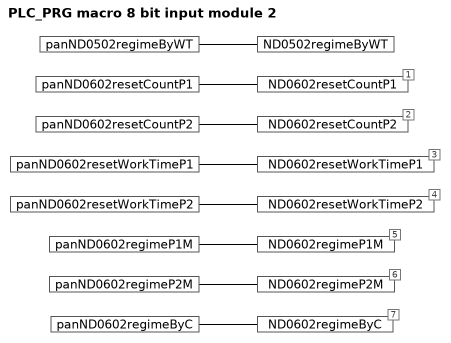
[picture p72: PLC_PRG macro 8 bit input module 2 (CFC)]
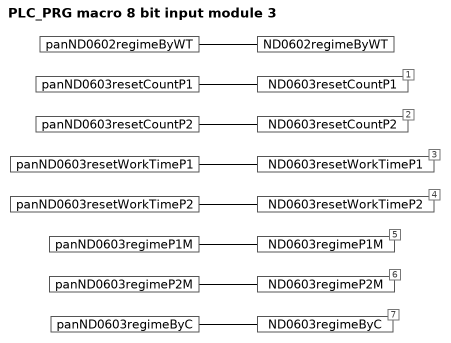
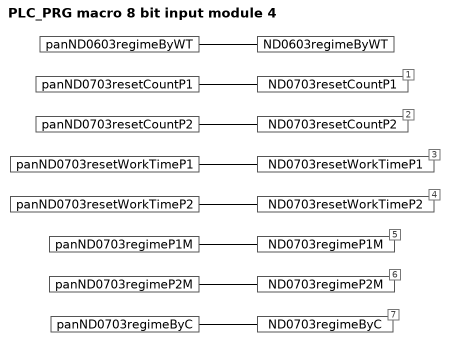
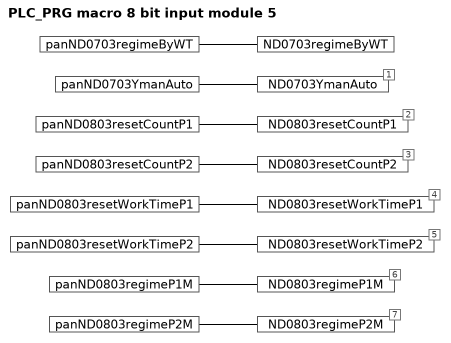
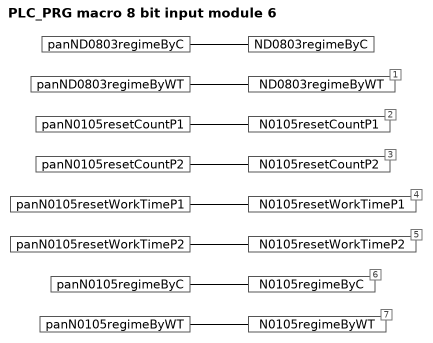
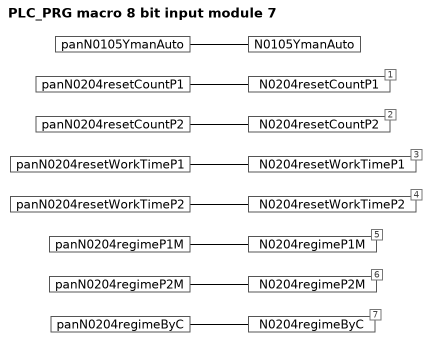
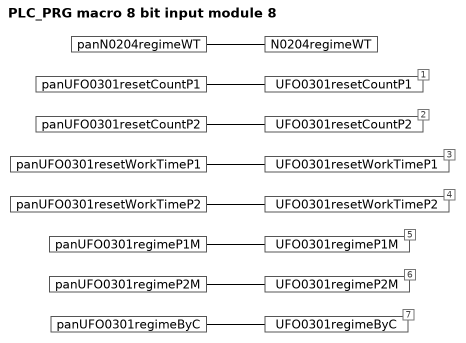
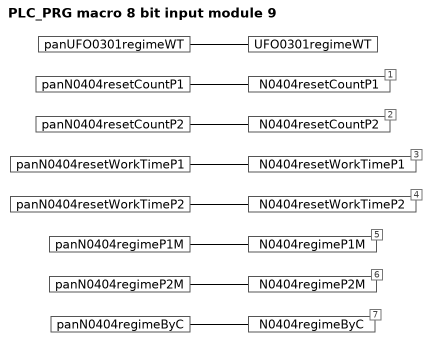
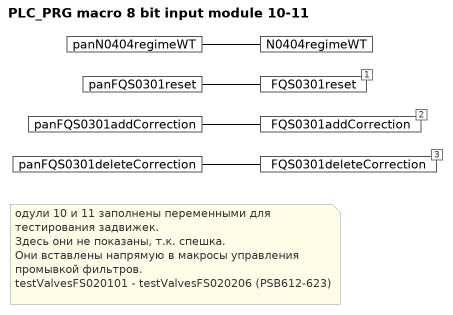
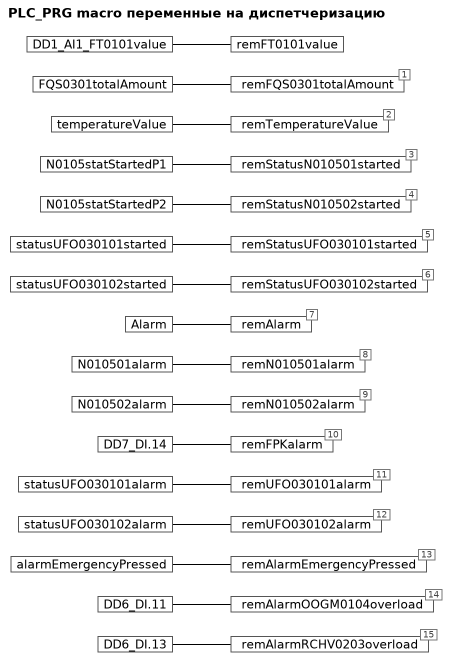
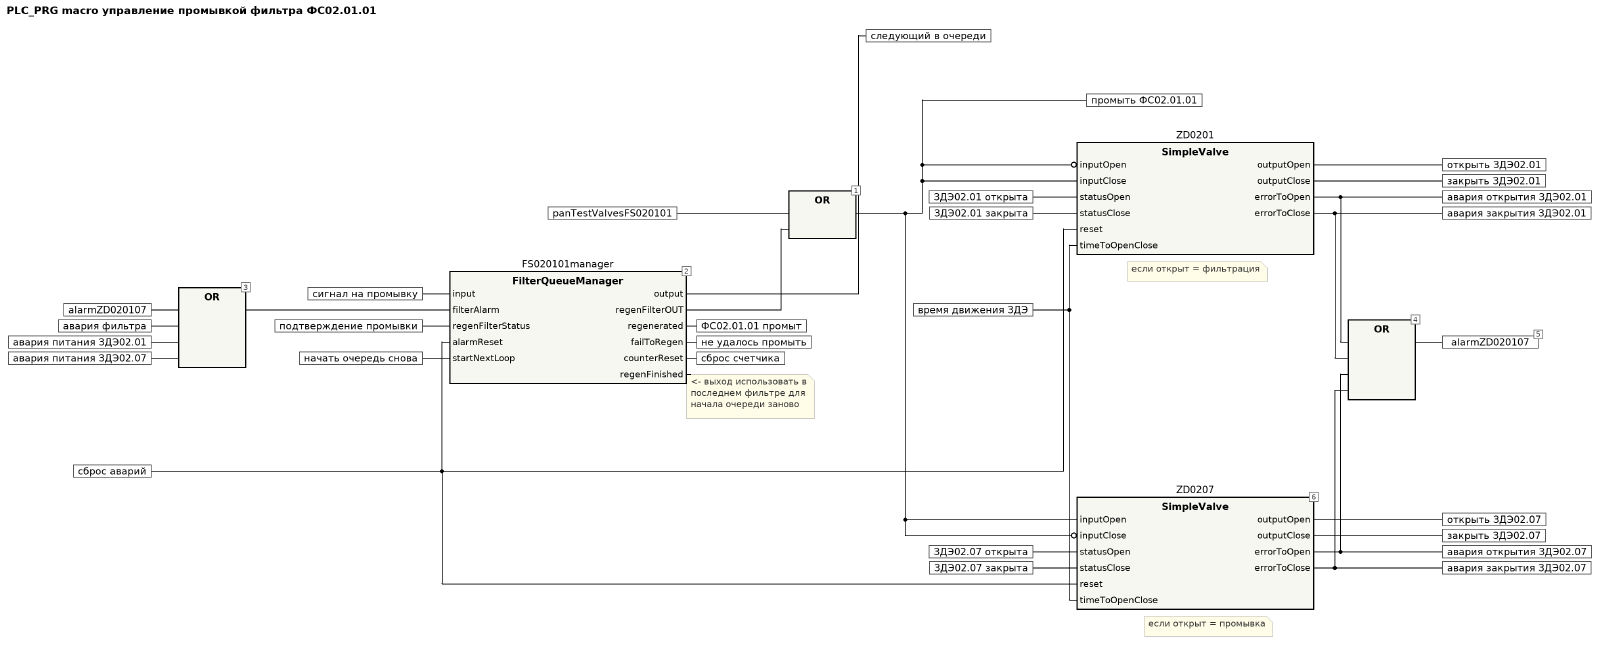
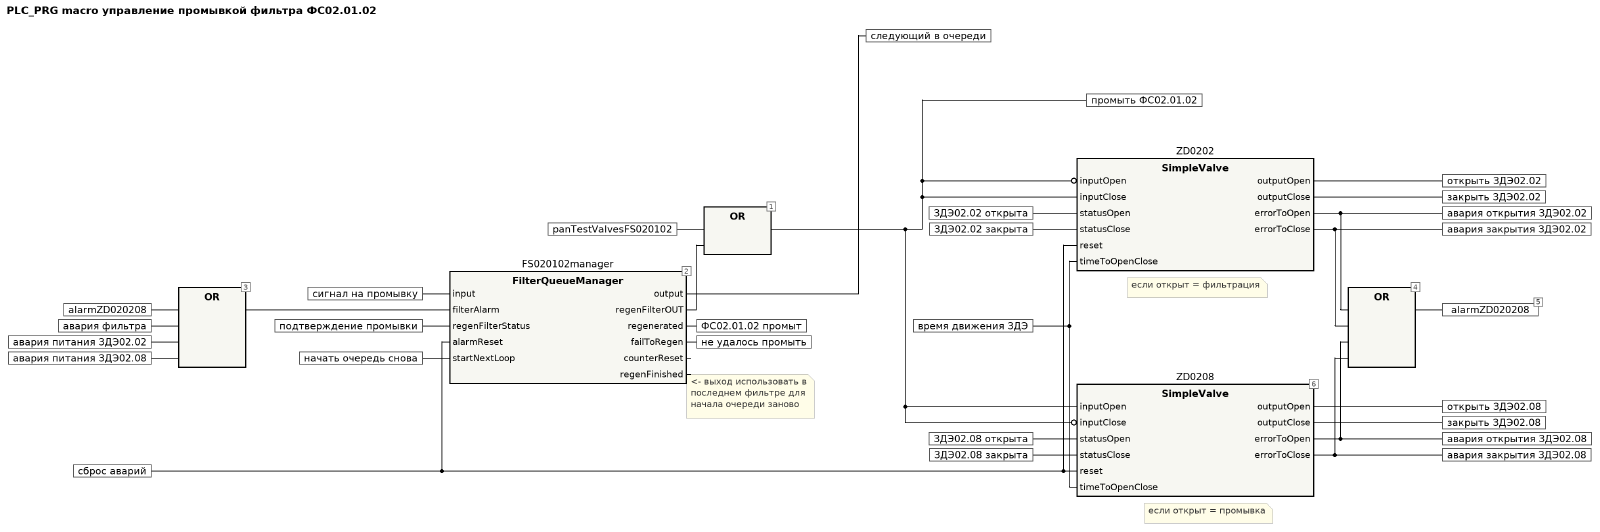
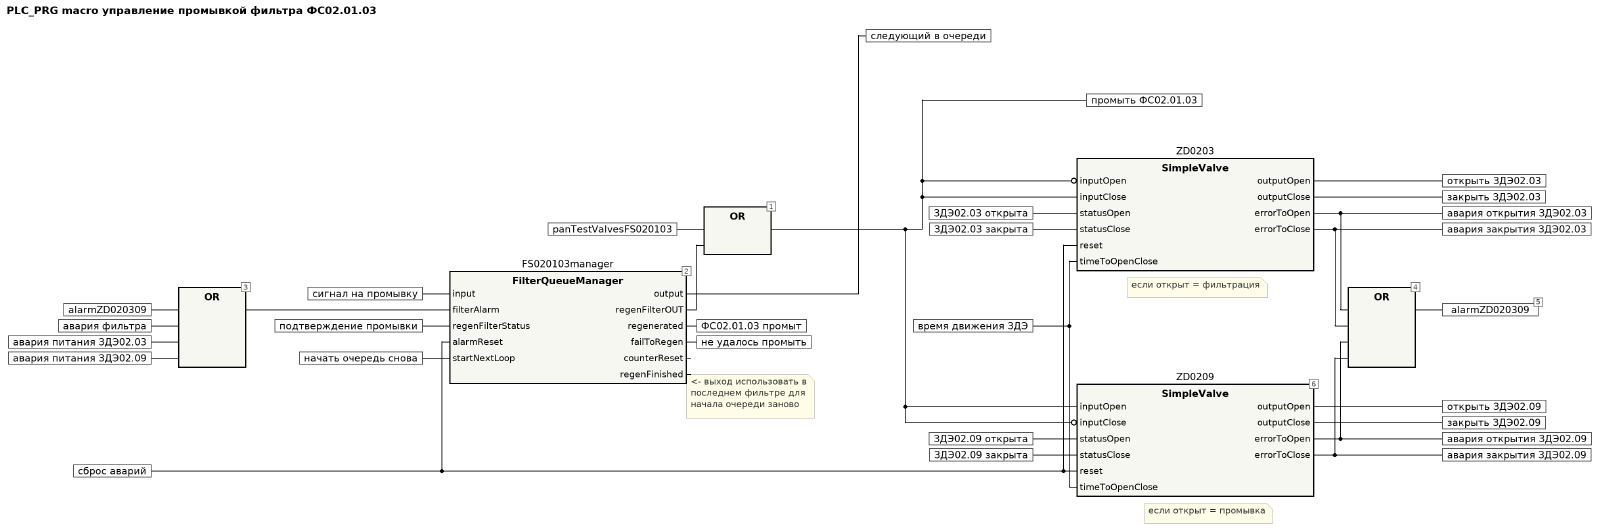
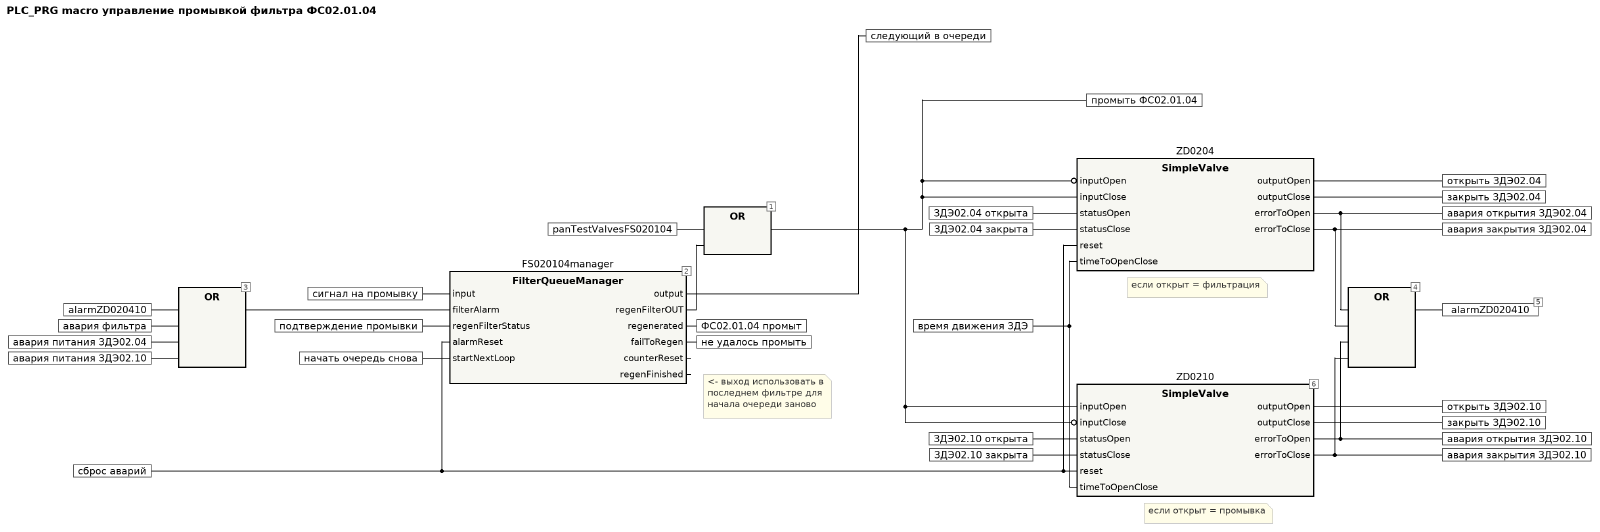
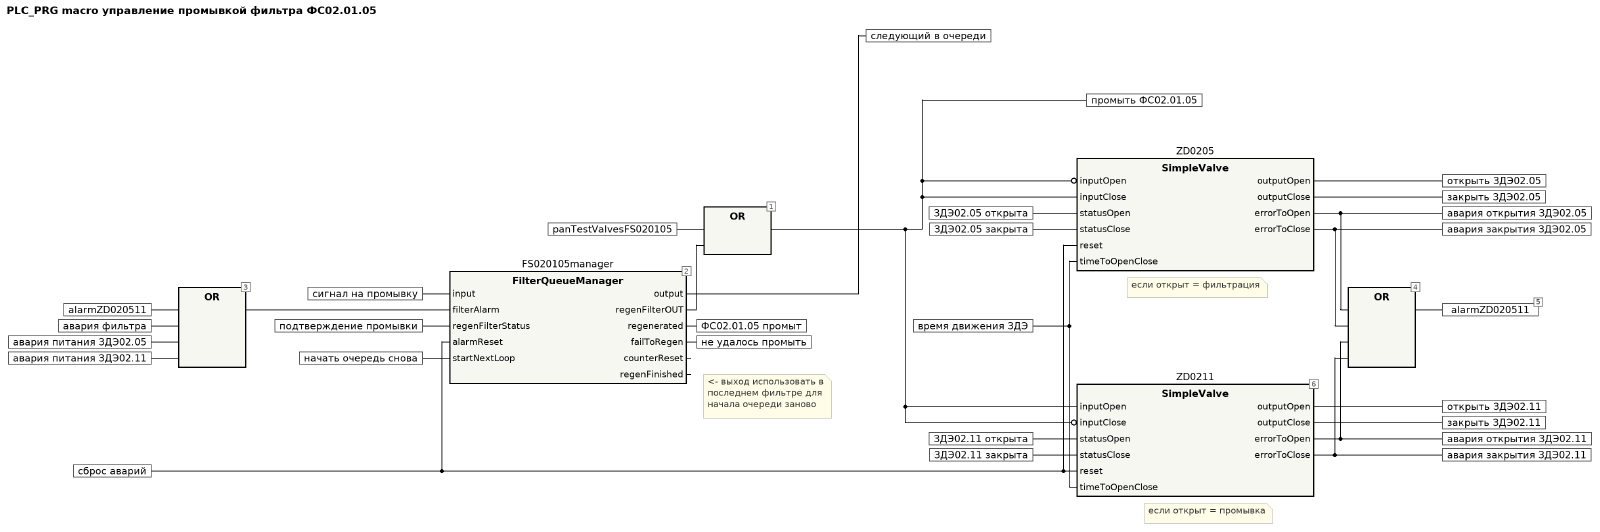
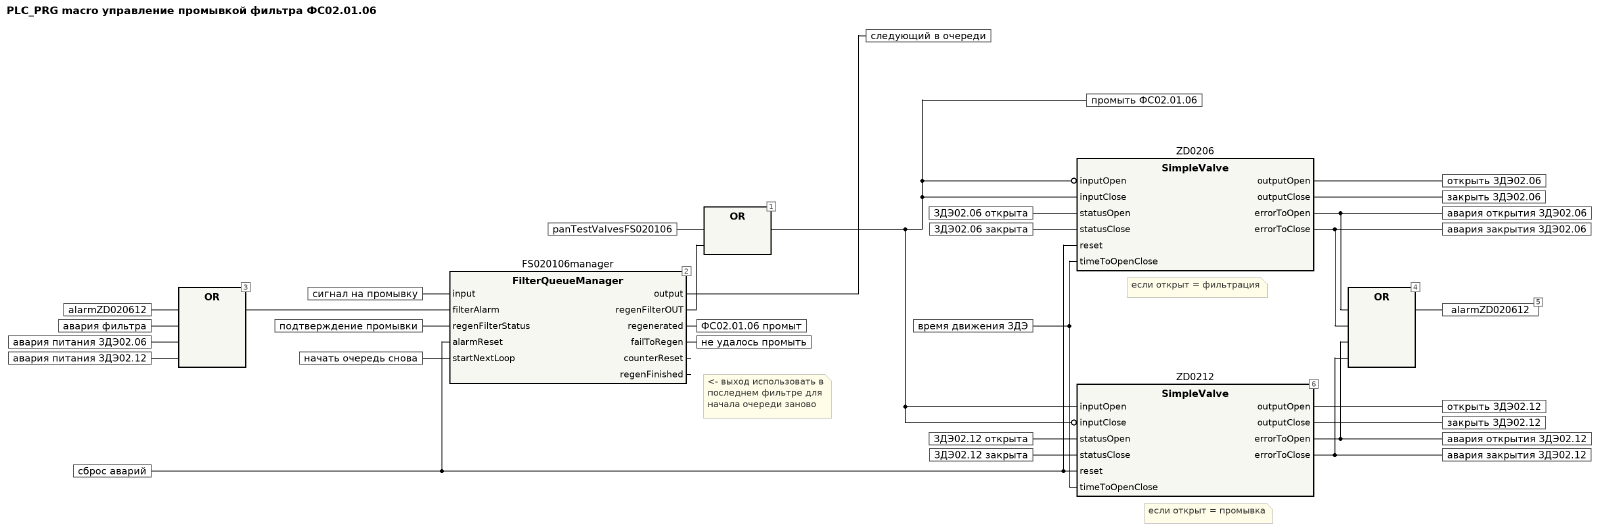
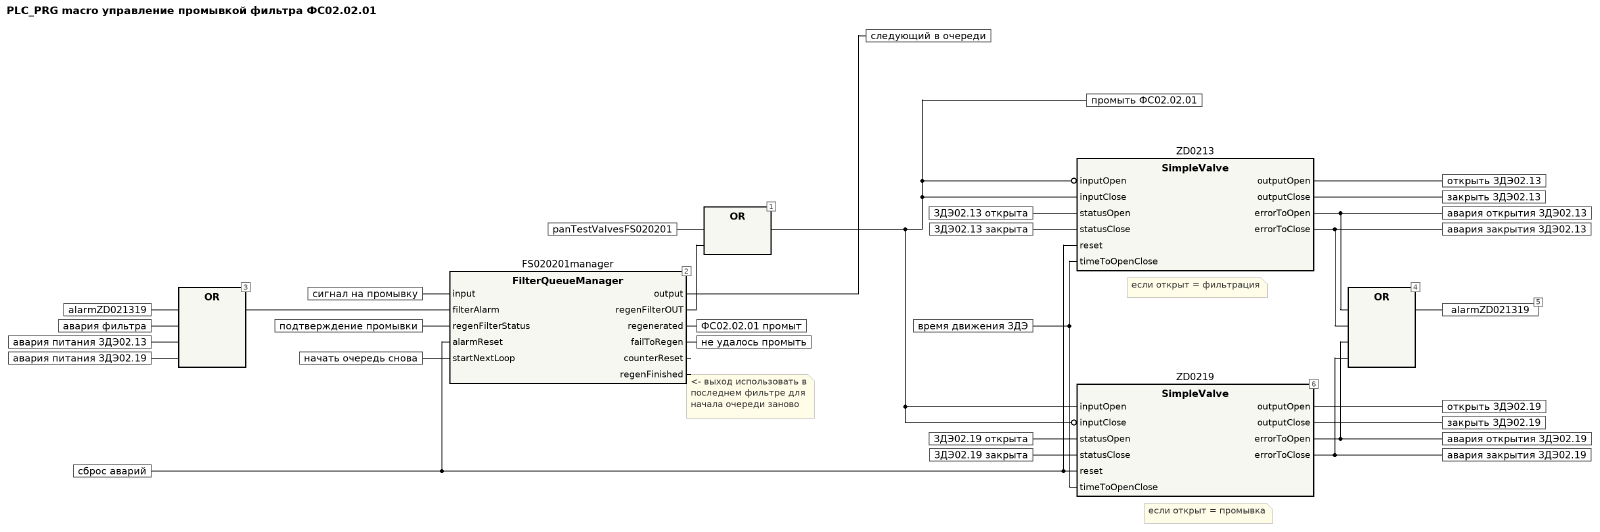
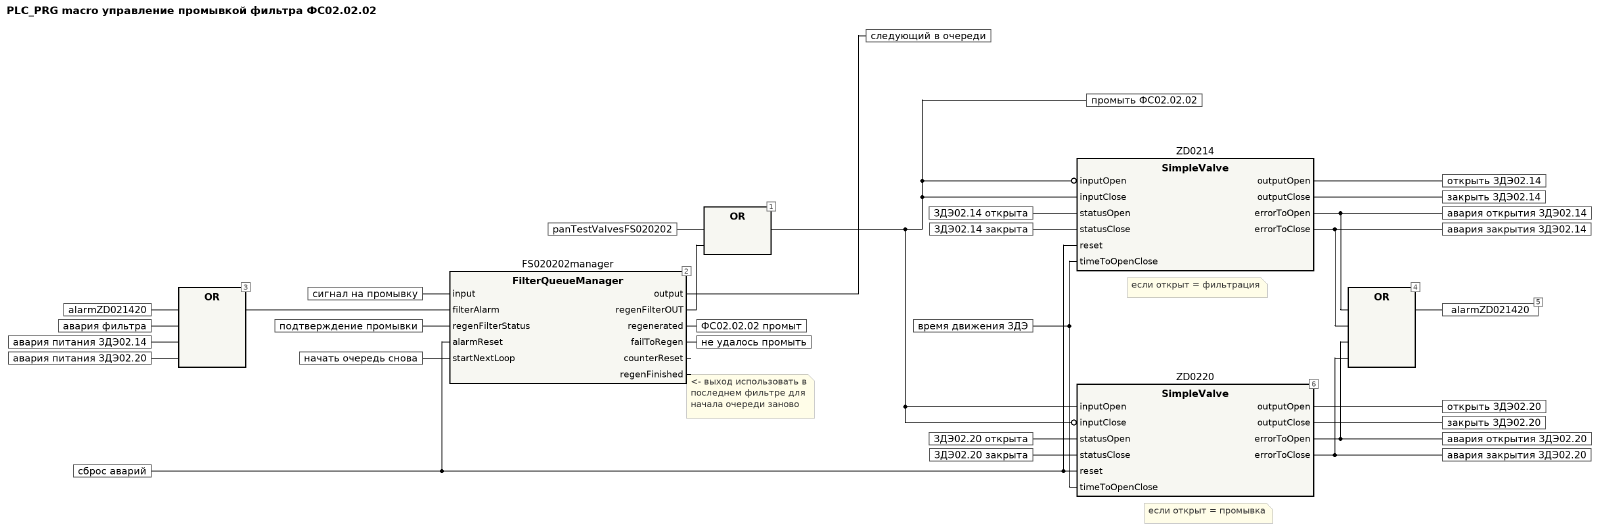
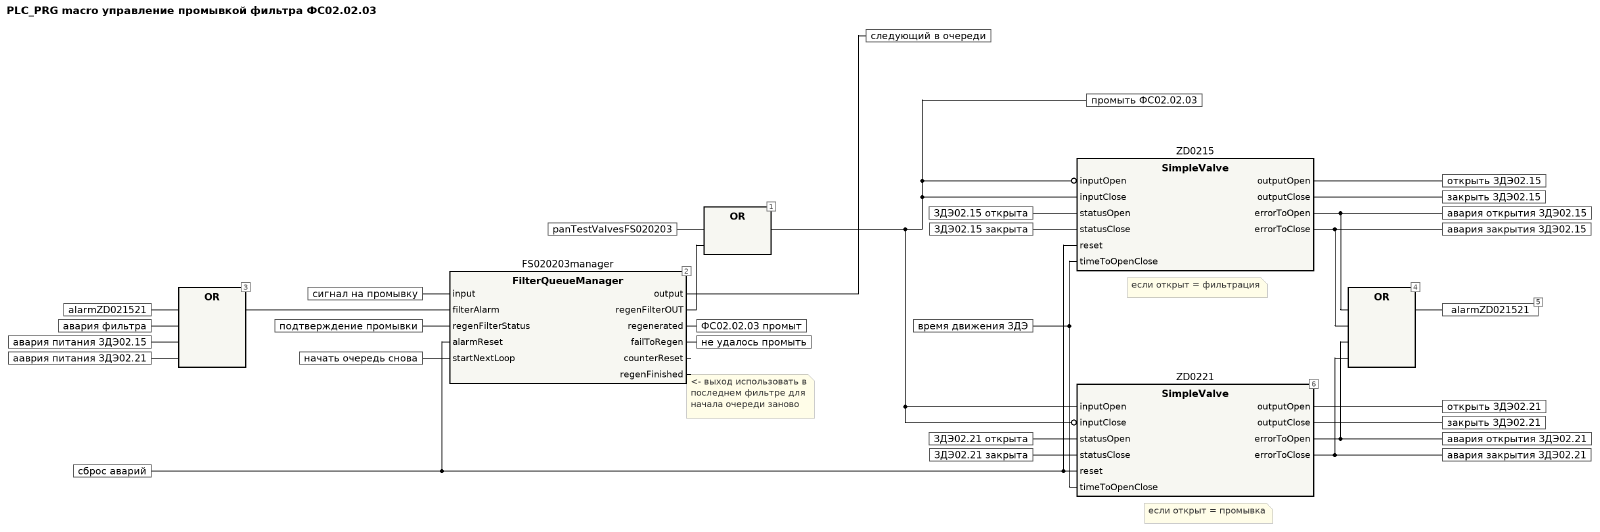
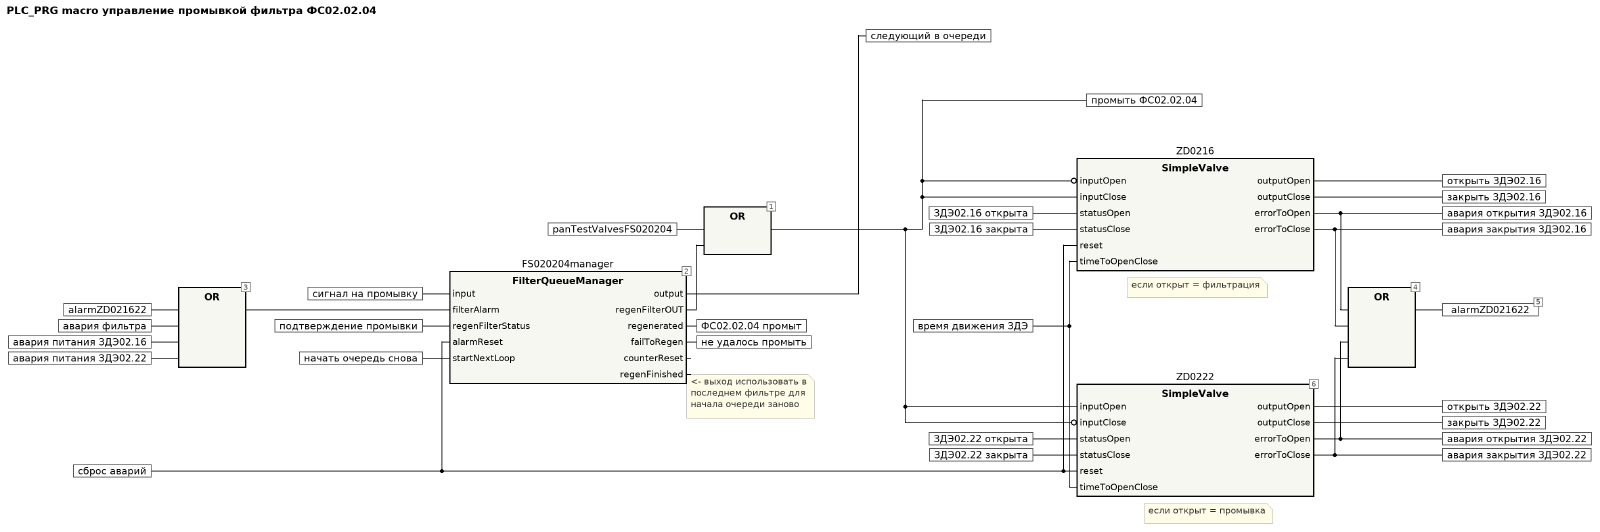
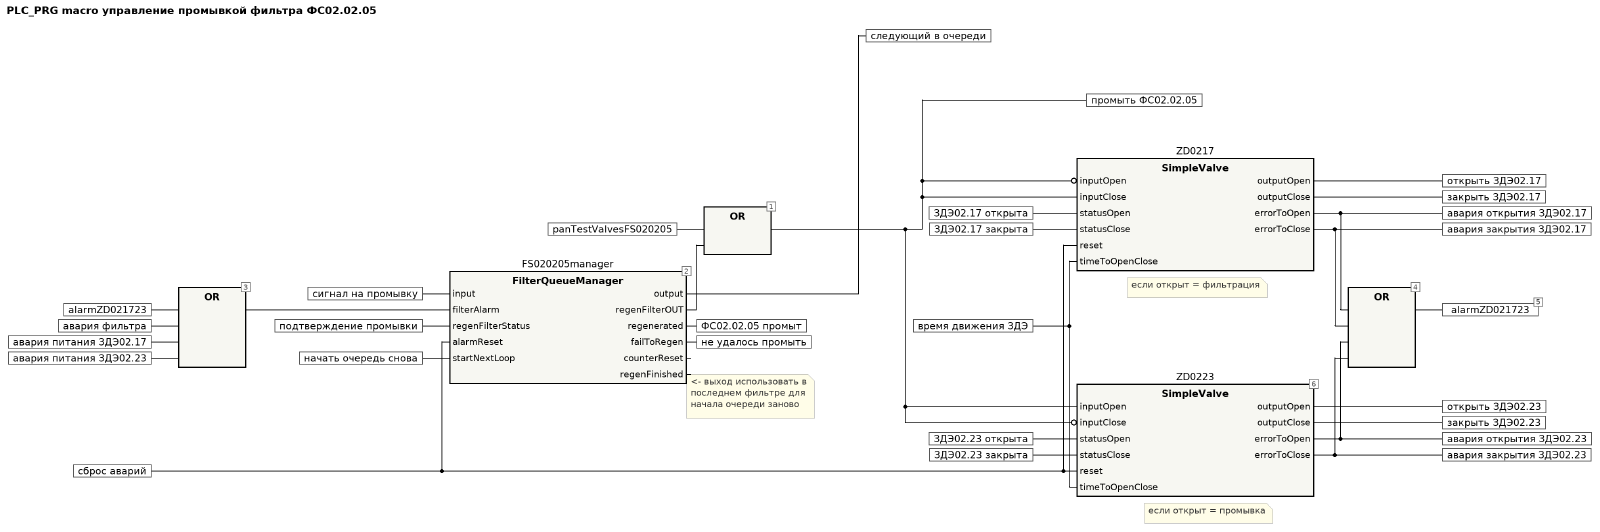
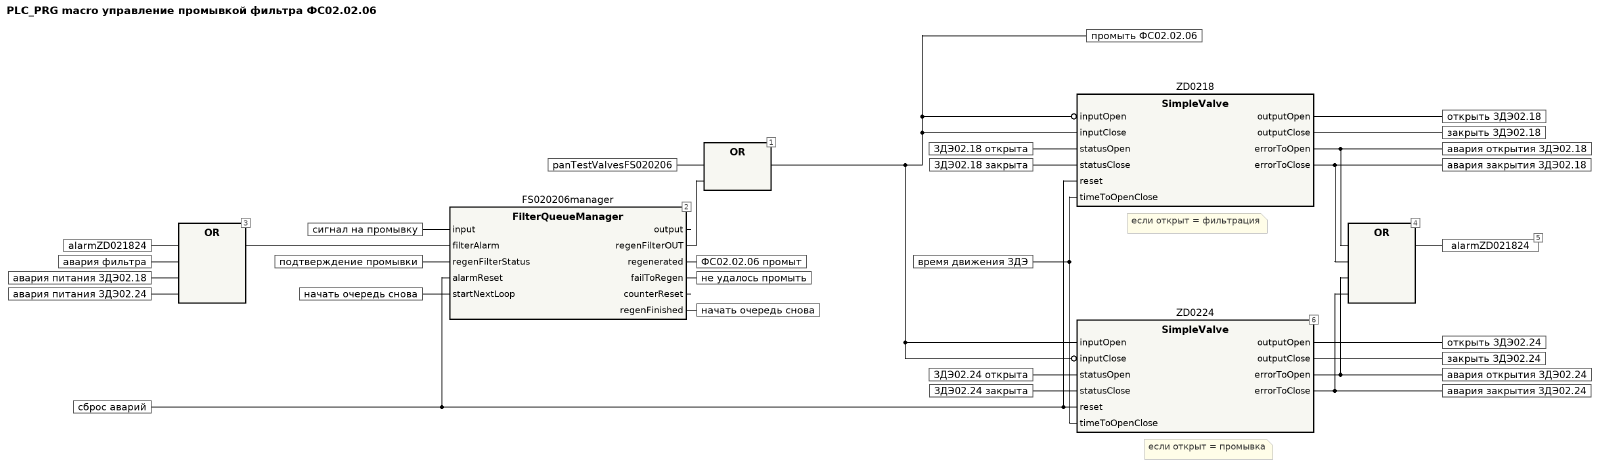
_CFC_ (* Continuous Function Chart, elements in execution order *)
(* в этом макросе лежит управление режимом тестирования задвижек ЗДЭ03 / Тестирование запрещает автоматический запуск УФО от ПЛК *)
(* 1=открыть; 0 = закрыть *)
(* авария питания КШЭ04.01 *)
(* авария НД05.02/02 *)
(* авария НД05.02/01 *)
(* инвертирование сигнала, чтобы все аварии / обозначались как 1 (TRUE) *)
(* авария питания ЗДЭ02.24 *)
(* авария питания ЗДЭ02.23 *)
(* авария питания ЗДЭ02.22 *)
(* авария питания ЗДЭ02.21 *)
(* авария питания ЗДЭ02.20 *)
(* авария питания ЗДЭ02.19 *)
(* авария питания ЗДЭ02.18 *)
(* авария питания ЗДЭ02.17 *)
(* авария питания ЗДЭ02.16 *)
(* авария питания ЗДЭ02.15 *)
(* авария питания ЗДЭ02.14 *)
(* авария питания ЗДЭ02.13 *)
(* авария питания ЗДЭ02.12 *)
(* авария питания ЗДЭ02.11 *)
(* авария питания ЗДЭ02.10 *)
(* авария питания ЗДЭ02.09 *)
(* авария питания ЗДЭ02.08 *)
(* авария питания ЗДЭ02.07 *)
(* авария питания ЗДЭ02.06 *)
(* авария питания ЗДЭ02.05 *)
(* авария питания ЗДЭ02.04 *)
(* авария питания ЗДЭ02.03 *)
(* авария питания ЗДЭ02.02 *)
(* авария питания ЗДЭ02.01 *)
(* очередь передается на 2 ступень *)
(* подсчет общего объема стоков, прошедшего через расходомер FT01.02 *)
(* сброс счетчика стоков до следующей промывки *)
(* авария (при 0) ФС02.02/01 *)
(* авария (при 0) ФС02.02/02 *)
(* авария (при 0) ФС02.02/03 *)
(* авария (при 0) ФС02.02/04 *)
(* авария (при 0) ФС02.02/05 *)
(* авария (при 0) ФС02.02/06 *)
(* авария (при 0) ФС02.01/01 *)
(* авария (при 0) ФС02.01/02 *)
(* авария (при 0) ФС02.01/03 *)
(* авария (при 0) ФС02.01/04 *)
(* авария (при 0) ФС02.01/05 *)
(* авария (при 0) ФС02.01/06 *)
(* 0=авария *)
(* заданный до промывки объем *)
(* текущий объем *)
(* Пуск Н02.04/02 *)
(* Пуск Н02.04/01 *)
(* Стоп Н02.04, / сброс самоподхвата реле, / если активно - пуск невозможен *)
(* Сухой ход Н02.04 (LS02.03) 0=сух.ход *)
(* Клапан КЭМ08.01 открыт. *)
(* Клапан КЭМ07.01 открыт. *)
(* Клапан КЭМ06.01 открыт. *)
(* Клапан КЭМ05.01 открыт. *)
(* промывка ФС02.02/01 *)
(* промывка ФС02.02/02 *)
(* промывка ФС02.02/03 *)
(* промывка ФС02.02/04 *)
(* промывка ФС02.02/05 *)
(* промывка ФС02.02/06 *)
(* Авария Н02.04/02 (0=авария) *)
(* Авария Н02.04/01 (0=авария) *)
(* импульсный расходомер *)
(* авария Н04.04/02, 0=авария *)
(* авария Н04.04/01, 0=авария *)
(* сухой ход Н04.04, 0=защита *)
(* авт.пуск Н04.04 *)
(* пуск Н04.04/01 *)
(* пуск Н04.04/02 *)
(* стоп Н04.04 *)
(* подающий насос ФПК работает *)
(* статус КШЭ04.01 закрыт *)
(* Закрыть КШЭ04.01 *)
(* статус КШЭ04.01 открыт *)
(* Открыть КШЭ04.01 *)
(* авария ФПК *)
(* Авария входа AI6 ПЛК, давл.ФПК *)
(* Давление на входе ФПК / 0...16 бар (мах допуст.10) *)
(* LSА02.01 Перелив РЧВ02.03 *)
(* авария питания ЗДЭ02.25 *)
(* термоконтакт Н01.05/02 *)
(* термоконтакт Н01.05/01 *)
(* Авария ЧРП Н01.05 *)
(* КМ3 питание насоса 2 *)
(* КМ2 питание насоса 1 *)
(* КМ1 питание ЧРП *)
(* Пуск  Н01.05 *)
(* время на создание потока *)
(* Стоп  Н01.05 (сброс самоподхвата реле) *)
(* SA1 Ручной выбор Н01.05/02 = главный *)
(* SA1 Ручной выбор Н01.05/01 = главный *)
(* LS01.04 - нижний уровень ОГМ01.04, сухой ход Н01.05 *)
(* LS01.03 - рабочий верхний уровень ОГМ01.04 автоматический пуск 01.05 *)
(* Статус ПУСК ЧРП Н01.05 *)
(* Инициализирует требуемые булевые переменные / в момент старта выполнения программы. *)
(* LSA01.02 перелив ОГМ01.04 *)
(* сухой ход НД08.03/02 *)
(* сухой ход НД08.03/01 *)
(* сухой ход НД08.03/02 *)
(* сухой ход НД08.03/01 *)
(* авария входа рН-метра QE01.02 *)
(* рН-метр QE01.01 на входе, / диапазон 0...14 *)
(* расходомер FT01.02 на входе, / диапазон 0...600куб/час *)
(* авария входа расходомера FT01.01 *)
(* управление 4...20мА НД08.04 *)
(* пуск/стоп НД08.04 *)
(* насос Н04.01 работает *)
(* авария НД08.04 *)
(* авария привода НД08.03/02 *)
(* авария привода НД08.03/01 *)
(* АВАРИИ *)
(* управление 4...20мА НД05.02/02 *)
(* пуск/стоп НД05.02/02 *)
(* авария НД05.02/02 *)
(* авария НД05.02/01 *)
(* пуск/стоп НД05.02/01 *)
(* управление 4...20мА НД05.02/01 *)
(* датчик температуры в помещении / (метран) диапазон: 0...+100С *)
(* лампа АВАРИЯ *)
(* авария входа датчика температуры *)
(* ошибка блока дозирования НД05.02 *)
(* авария НД06.02/02 *)
(* авария НД06.02/01 *)
(* управление 4...20мА НД06.02/02 *)
(* пуск/стоп НД06.02/02 *)
(* пуск/стоп НД06.02/01 *)
(* управление 4...20мА НД06.02/01 *)
(* авария НД06.03/02 *)
(* авария НД06.03/01 *)
(* управление 4...20мА НД06.03/02 *)
(* пуск/стоп НД06.03/02 *)
(* пуск/стоп НД06.03/01 *)
(* управление 4...20мА НД06.03/01 *)
(* авария НД06.02/02 *)
(* авария НД06.02/01 *)
(* авария НД06.03/02 *)
(* авария НД06.03/01 *)
(* авария НД07.03/02 *)
(* авария НД07.03/01 *)
(* пуск/стоп НД07.03/02 *)
(* пуск/стоп НД07.03/01 *)
(* управление 4...20мА НД07.03/02 *)
(* управление 4...20мА НД07.03/01 *)
(* авария НД07.03/02 *)
(* авария НД07.03/01 *)
(* авария привода НД08.03/02 *)
(* авария привода НД08.03/01 *)
(* управление 4...20мА НД08.03/02 *)
(* пуск/стоп НД08.03/02 *)
(* пуск/стоп НД08.03/01 *)
(* управление 4...20мА НД08.03/01 *)
(* авария НД08.04 *)
(* расходомер FT01.01 на входе, / диапазон 0...600куб/час *)
(* авария входа расходомера FT01.02 *)
(* авария входа рН-метра QE01.01 *)
(* рН-метр QE01.02 на входе, / диапазон 0...14 *)
(* ФПК не запустился *)
(* ФПК готов к приему *)
(* подающий насос ФПК работает *)
(* авария ФПК *)
(* Давление на входе ФПК (0...16 бар) *)
(* датчик уровня осадка *)
(* Защита от сухого хода насоса ФПК *)
(* запуск фильтрации *)
(* время работы ФПК после спада сигнала датч.осадка *)
(* время контроля старта ФПК (по умолч.=3мин) *)
(* авария Н04.04/02 *)
(* авария Н04.04/01 *)
(* авария УФО03.01/01 *)
(* авария УФО03.01/02 *)
(* работа УФО03.01/01 *)
(* Для подачи предостережения на пульте / оператора (при необходимости), а также / сигнализации лампой АВАРИЯ. *)
(* авария УФО03.01/01 *)
(* работа УФО03.01/02 *)
(* авария УФО03.01/02 *)
(* Контроль, если УФО включили вручную, / а потока при этом нет. *)
(* работа М06.04 (УПК) *)
(* работа М07.02 (УПЩ) *)
(* работа М08.02 (УПФ) *)
(* авария М06.04 (УПК) *)
(* авария М07.02 (УПЩ) *)
(* авария М08.02 (УПФ) *)
(* пуск/стоп НД07.03/02 *)
(* пуск/стоп НД07.03/01 *)
(* пуск/стоп НД08.04 *)
(* пуск/стоп НД06.02/02 *)
(* пуск/стоп НД06.02/01 *)
(* пуск/стоп НД06.03/02 *)
(* пуск/стоп НД06.03/01 *)
(* пуск/стоп НД08.03/02 *)
(* пуск/стоп НД08.03/01 *)
(* промывка ФС02.01/01 *)
(* промывка ФС02.01/02 *)
(* промывка ФС02.01/03 *)
(* промывка ФС02.01/04 *)
(* промывка ФС02.01/05 *)
(* промывка ФС02.01/06 *)
(* Авария Н02.04/02 (0=авария) *)
(* Авария Н02.04/01 (0=авария) *)
(* здесь мгновенный расход / в кубометрах в час (FT01.02) *)
(* выдает импульс / каждую секунду *)
(* если есть расход / (больше нуля) *)
(* преобразуем расход из / кубометров в час в / кубометры в секунду *)
(* суммируем каждую секунду значение / мгновенного расхода в кубометрах в секунду *)
(* блок подачи сигнала на промывку *)
(* авария КНС *)
(* Авария питания розеток / управл.клапанов фильтров. *)
(* Авария питания клапанов КЭМ. *)
(* авария сети (РКФ) *)
(* Блок управления разрешением работы КНС *)
(* Нажат аварийный стоп. *)
(* разрешение работы КНС / 1 = разрешено *)
(* авария сети (РКФ) *)
(* Нажат аварийный стоп. *)
(* LSA01.02 перелив ОГМ01.04 *)
(* контроль обрыва или ошибок модулей в сети ПЛК *)
(* вкл КМ2 *)
(* статус-пуск Н01.05/01 *)
(* Статус ПУСК / ЧРП Н01.05 *)
(* вкл КМ3 *)
(* статус-пуск Н01.05/02 *)
(* авария питания ЗДЭ03.01 *)
(* авария питания ЗДЭ03.02 *)
(* авария обоих УФО, если проблемы / открытия/закрытия на одной из задвижек *)
(* 0 = перелив *)
#0 rTrigStartInitializer:R_TRIG(CLK: TRUE)
#1 startInitializer <= #0.Q
#2 MACRO контроль температуры в помещении(pin 1 "вход датчика температуры": DD1_AI0, pin 2 "минимально допустимая температура в помещении": maxTemperature, pin 3 "максимально допустимая температура в помещении": minTemperature)
	(* не смотрим конкретный тип ошибки / (работает не точно, обрыв определяет как слишком маленькое значение) / если не равно 0 - значит на входе ошибка *)
	(* задаем границы допустимой температуры в помещении / проверяем что измеренное значение в заданном диапазоне *)
	#3 DD1_AI0_temperature:DECODE_FLOAT(VALUE: pin 1, DEF_VALUE: -)
	#4 NE(#3._ERR, 0)
	out 2 "авария датчика температуры" <= #4
	out 1 "температура в помещении" <= #3.OUT_VALUE
	#5 REAL_TO_INT(#3.OUT_VALUE)
	#6 temperatureLimits:LIMITALARM(IN: #5, HIGH: pin 3, LOW: pin 2)
	out 3 "температура выше заданного диапазона" <= #6.O
	out 4 "температура ниже заданного диапазона" <= #6.U
	#7 temperatureLimits:LIMITALARM(IN: -, HIGH: -, LOW: -)
END_MACRO
#8 temperatureValue <= #2.out 1
#9 DD1_AI0_error <= #2.out 2
#10 alarmHighTemperature <= #2.out 3
#11 alarmLowTemperature <= #2.out 4
#12 OR(testKSHE0401, DD7_DI.13)
#13 MACRO клапан шаровый перед ФПК (КШЭ04.01)(pin 1 "сигнал "подающий насос ФПК" работает": #12, pin 2 "статус КШЭ04.01 открыт": DD9_DI.2, pin 3 "статус КШЭ04.01 закрыт": DD9_DI.3, pin 4 "сброс аварий": alarmReset, pin 5 "время на открытие/закрытие": timeToOpenCloseValve)
	#14 FPKkshe0401DelayToOpen:TON(IN: #16.outputOpen, PT: T#1s)
	out 1 "выход на открытие КШЭ04.01" <= #14.Q
	#15 FPKkshe0401DelayToClose:TON(IN: #16.outputClose, PT: T#1s)
	out 2 "выход на закрытие КШЭ04.01" <= #15.Q
	#16 FPKkshe0401:SimpleValve(inputOpen: pin 1, inputClose: #17, statusOpen: pin 2, statusClose: pin 3, reset: pin 4, timeToOpenClose: pin 5)
	#17 NOT(pin 1)
	out 3 "авария на открытие КШЭ04.01" <= #16.errorToOpen
	out 4 "авария на закрытие КШЭ04.01" <= #16.errorToClose
END_MACRO
#18 DD4_DO.2 <= #13.out 1
#19 DD4_DO.3 <= #13.out 2
#20 FPKkshe0401errorToOpen <= #13.out 3
#21 FPKkshe0401errorToClose <= #13.out 4
#22 OR(DD1_AI0_error, DD1_AI1_error, DD1_AI2_error, DD1_AI3_error, DD1_AI4_error, alarmHighTemperature, alarmLowTemperature, ND0502dosingError, ND0602dosingError, ND0603dosingError, ND0803dosingError, ND0804dosingError, DD1_DI6, DD1_DI7, N010501alarm, N010502alarm, ZDE0225errorToOpen, ZDE0225errorToClose, DD7_DI.14, FPKnotStarted, DD1_AI5_error, FPKkshe0401errorToOpen, FPKkshe0401errorToClose, DD5_DI.27, DD5_DI.29, filterFailToRegen020101, errorToOpenZD0201, errorToCloseZD0201, errorToOpenZD0207, errorToCloseZD0207, filterFailToRegen020102, errorToOpenZD0202, errorToCloseZD0202, errorToOpenZD0208, errorToCloseZD0208, filterFailToRegen020103, errorToOpenZD0203, errorToCloseZD0203, errorToOpenZD0209, errorToCloseZD0209, filterFailToRegen020104, errorToOpenZD0204, errorToCloseZD0204, errorToOpenZD0210, errorToCloseZD0210, filterFailToRegen020105, errorToOpenZD0205, errorToCloseZD0205, errorToOpenZD0211, errorToCloseZD0211, filterFailToRegen020106, errorToOpenZD0206, errorToCloseZD0206, errorToOpenZD0212, errorToCloseZD0212, filterFailToRegen020201, errorToOpenZD0213, errorToCloseZD0213, errorToOpenZD0219, errorToCloseZD0219, filterFailToRegen020202, errorToOpenZD0214, errorToCloseZD0214, errorToOpenZD0220, errorToCloseZD0220, filterFailToRegen020203, errorToOpenZD0215, errorToCloseZD0215, errorToOpenZD0221, errorToCloseZD0221, filterFailToRegen020204, errorToOpenZD0216, errorToCloseZD0216, errorToOpenZD0222, errorToCloseZD0222, filterFailToRegen020205, errorToOpenZD0217, errorToCloseZD0217, errorToOpenZD0223, errorToCloseZD0223, filterFailToRegen020206, errorToOpenZD0218, errorToCloseZD0218, errorToOpenZD0224, errorToCloseZD0224, alarmPLKnetwork, alarmND050201, alarmND050202, alarmND060201, alarmND060202, alarmND060301, alarmND060302, alarmND070301, alarmND070302, alarmND080301, alarmND080302, alarmND0804, alarmOGM0104overload, alarmRCHV0203overload, alarmN040402, alarmN040401, alarmM0604, alarmM0702, alarmM0802, alarmN020401, alarmN020402, alarmFS020101, alarmFS020102, alarmFS020103, alarmFS020104, alarmFS020105, alarmFS020106, alarmFS020201, alarmFS020202, alarmFS020203, alarmFS020204, alarmFS020205, alarmFS020206, alarmZDE0201power, alarmZDE0202power, alarmZDE0203power, alarmZDE0204power, alarmZDE0205power, alarmZDE0206power, alarmZDE0207power, alarmZDE0208power, alarmZDE0209power, alarmZDE0210power, alarmZDE0211power, alarmZDE0212power, alarmZDE0213power, alarmZDE0214power, alarmZDE0215power, alarmZDE0216power, alarmZDE0217power, alarmZDE0218power, alarmZDE0219power, alarmZDE0220power, alarmZDE0221power, alarmZDE0222power, alarmZDE0223power, alarmZDE0224power, alarmZDE0225power, alarmKSHE0401power, alarmKNS, alarmPowerSocketFS, alarmKEMvalvesPower, alarmEmergencyPressed, alarmRKF, errorToOpenZDE0301, errorToCloseZDE0301, errorToOpenZDE0302, errorToCloseZDE0302, alarmZDE0301power, alarmZDE0302power)
#23 DD1_DO11 <= #22
#24 alarm <= #22
#25 MACRO контроль аналогового входа DD1_AI1(pin 1 "вход": DD1_AI1)
	(* Не смотрим конкретную ошибку, / определяем,что вход неисправен без расшифровки. *)
	#26 DD1_AI1_FT0101:DECODE_FLOAT(VALUE: pin 1, DEF_VALUE: -)
	#27 NE(#26._ERR, 0)
	out 2 "авария" <= #27
	out 1 "выход" <= #26.OUT_VALUE
END_MACRO
#28 DD1_AI1_FT0101value <= #25.out 1
#29 DD1_AI1_error <= #25.out 2
#30 MACRO контроль аналогового входа DD1_AI2(pin 1 "вход": DD1_AI2)
	(* Не смотрим конкретную ошибку, / определяем,что вход неисправен без расшифровки. *)
	#31 DD1_AI2_FT0102:DECODE_FLOAT(VALUE: pin 1, DEF_VALUE: -)
	#32 NE(#31._ERR, 0)
	out 2 "авария" <= #32
	out 1 "выход" <= #31.OUT_VALUE
END_MACRO
#33 DD1_AI2_FT0102value <= #30.out 1
#34 DD1_AI2_error <= #30.out 2
#35 MACRO управление Н01.05 (поддержание заданного расхода по FT01.02)(pin 1 "статус ПУСК ЧРП (реле)": DD5_DI.4, pin 2 "LS01.03 раб.уров.": DD6_DI.12, pin 3 "LS01.04 ниж.уров.(сух.ход)": DD5_DI.0, pin 4 "SA1ручной выб.Н01.05/01-главный": DD5_DI.5, pin 5 "SA1ручной выб.Н01.05/02-главный": DD5_DI.6, pin 6 "включить режим "по кол.вкл."": N0105regimeByC, pin 7 "включить режим "по наработке"": N0105regimeByWT, pin 8 "значение расхода от FT01.02": DD1_AI2_FT0102value, pin 9 "уставка расхода": N0105flowSetValue, pin 10 "время на создание потока": N0105minFlowTime, pin 11 "Р-коэфф.": N0105koeffP, pin 12 "I-коэфф": N0105koeffI, pin 13 "Д-коэфф": N0105koeffD, pin 14 "управление ЧРП в ручн.реж.(4...20мА)": N0105YoutManual, pin 15 "переключатель управление ЧРП РУЧН/АВТ": N0105YmanAuto, pin 16 "мин.допустимый расход": N0105minFlow, pin 17 "термоконтакт Н01.05/01": DD5_DI.2, pin 18 "термоконтакт Н01.05/02": DD5_DI.3, pin 19 "авария ЧРП Н01.05": DD5_DI.1, pin 20 "сброс аварии": alarmReset, pin 21 "сброс кол-ва вкл.Н01.05/01": N0105resetCountP1, pin 22 "сброс кол-ва вкл.Н01.05/02": N0105resetCountP2, pin 23 "сброс наработки Н01.05/01": N0105resetWorkTimeP1, pin 24 "сброс наработки Н01.05/02": N0105resetWorkTimeP2)
	(* Если насос создает давление меньше / указанного, то авария. *)
	(* если на входе true / то нижнее значение, / иначе то, что посередине *)
	(* по умолчанию при старте программы *)
	(* управление Н01.05 - поддержание / заданного расхода по FT01.02 *)
	(* режимы по количеству включений,  или по наработке / активны если оба входа SA1 не активны *)
	(* Пуск  Н01.05 *)
	(* время на создание потока *)
	#36 OR(pin 2, #37.Q)
	#37 N0105startTrig:R_TRIG(CLK: pin 1)
	#38 N0105stopTrig:F_TRIG(CLK: pin 1)
	#39 N0105startTrigg:RS(SET: #36, RESET1: #42)
	#40 N0105regime:choosePumpRegime(start: #39.Q1, pump1Main: pin 4, pump2Main: pin 5, byCounter: #49, byWorkTime: #54)
	out 2 "статус режим "Н01.05/01 - главный"" <= #40.pump1MainActive
	out 3 "статус режим "Н01.05/02 - главный"" <= #40.pump2MainActive
	#41 AND(#53.pump1active, #63)
	out 4 "статус режим "по кол-ву вкл."" <= #40.byCounterActive
	out 15 "авария Н01.05/01" <= #45.Q1
	#42 OR(#38.Q, #43)
	out 5 "статус режим "по наработке"." <= #40.byWorkTimeActive
	#43 NOT(pin 3)
	#44 OR(#41, #48, NOT pin 17)
	#45 N010501alarmTrig:RS(SET: #44, RESET1: pin 20)
	#46 N010501alarm <= #45.Q1
	#47 NOT(#39.Q1)
	out 1 "СТОП (сброс самоподхвата реле пуска ЧРП)." <= #47
	#48 AND(#53.pump1active, NOT pin 19)
	#49 AND(NOT pin 4, NOT pin 5, #52.Q1)
	#50 OR(pin 6, startInitializer)
	#51 N0105regByCinit:R_TRIG(CLK: #50)
	#52 N0105regByCtrig:RS(SET: #51.Q, RESET1: #55.Q)
	#53 N0105twoPumpOneDriveManager:TwoPumpOneDriveManager(startStopPump1: #40.startPump1, startStopPump2: #40.startPump2, alarmPump1: N010501alarm, alarmPump2: N010502alarm, alarmReset: alarmReset, counterStart: #40.startByCounter, Pump1ResetCounter: pin 21, Pump2ResetCounter: pin 22, ValueToResetCounter: -, workTimeStart: #40.startByWorkTime, workTimePump1Reset: pin 23, workTimePump2Reset: pin 24, timeKM1off: -, timeKM23DelayON: -, timeKM23offDelay: -, timeReadyToStartDelay: -)
	out 6 "кол-во включений Н01.05/01" <= #53.counterPump1
	out 7 "кол-во включений Н01.05/02" <= #53.counterPump2
	out 8 "наработка Н01.05/01" <= #53.currentWorkTimePump1
	#54 AND(NOT pin 4, NOT pin 5, #56.Q1)
	out 9 "наработка Н01.05/02" <= #53.currentWorkTimePump2
	out 10 "КМ1-питание ЧРП" <= #53.DriveKM
	#55 N0105regWTinit:R_TRIG(CLK: pin 7)
	#56 N0105regWTtrig:RS(SET: #55.Q, RESET1: #51.Q)
	out 11 "КМ2-питание Н01.05/01" <= #53.pump1KM
	out 12 "КМ3-питание Н01.05/02" <= #53.pump2KM
	out 13 "пуск ЧРП (Н01.05)" <= #53.driveStart
	out 16 "авария Н01.05/02" <= #59.Q1
	#57 AND(NOT pin 19, #53.pump2active)
	#58 OR(#57, #61, NOT pin 18)
	#59 N010502alarmTrig:RS(SET: #58, RESET1: pin 20)
	#60 N010502alarm <= #59.Q1
	#61 AND(#53.pump2active, #63)
	#62 N0105timerminFlow:TON(IN: #53.driveStart, PT: pin 10)
	#63 AND(#62.Q, #64)
	#64 LE(pin 8, pin 16)
	#65 SEL(#53.driveStart, 0, #66.Y)
	out 14 "управление ЧРП (4...20мА)" <= #65
	#66 N0105pidReg:PID(ACTUAL: pin 8, SET_POINT: pin 9, KP: pin 11, TN: pin 12, TV: pin 13, Y_MANUAL: pin 14, Y_OFFSET: -, Y_MIN: 4, Y_MAX: 20, MANUAL: pin 15, RESET: #66.OVERFLOW)
END_MACRO
#67 DD4_DO.13 <= #35.out 1
#68 N0105statRegimeP1M <= #35.out 2
#69 N0105statRegimeP2M <= #35.out 3
#70 N0105statRegimeByC <= #35.out 4
#71 N0105statRegimeByWT <= #35.out 5
#72 N0105counterP1 <= #35.out 6
#73 N0105counterP2 <= #35.out 7
#74 N0105workTimeP1 <= #35.out 8
#75 N0105workTimeP2 <= #35.out 9
#76 DD2_DO.0 <= #35.out 10
#77 DD2_DO.1 <= #35.out 11
#78 DD2_DO.2 <= #35.out 12
#79 DD1_DO0 <= #35.out 13
#80 DD1_AO0 <= #35.out 14
#81 N010501alarm <= #35.out 15
#82 N010502alarm <= #35.out 16
#83 MACRO Сигналы работы с ФП04.02 (фильтр-пресс)(pin 1 "датчик уровня осадка": DD7_DI.15, pin 2 "время работы ФПК (после выкл.датч.осадка)": FPKtimeToWork, pin 3 "защита от сухого хода": DD6_DI.10, pin 4 "ошибка входа AI (обрыв)": DD1_AI5_error, pin 5 "авария ФПК": DD7_DI.14, pin 6 "фильтр-пресс готов к приему": DD7_DI.12, pin 7 "давление на входе в ФПК": DD1_AI5_FPKpressureValue, pin 8 "мах допустимое давление": FPKmaxPressureValue, pin 9 "подающий насос ФПК работает": DD7_DI.13, pin 10 "время контроля старта ФПК": FPKnotStartedTime, pin 11 "сброс аварий": alarmReset)
	(* Условие сброса сигнала о грязном фильтр-прессе: / 1. Пропал сигнал о готовности ФПК; / 2. Появился сигнал о готовности ФПК. / Это значит, что оператор раздвигал плиты, / чистил и снова сдвигал их. *)
	(* максимально допустимое давление / на входе ФПК *)
	(* Давление на входе ФПК / 0...16 бар (мах допуст.10) *)
	(* Время работы ФПК после / спада сигнала уровня осадка / по умолч.15мин. *)
	(* LES01.01-сигнал датчика уровня осадка ОГМ01.04 / запуск процесса фильтрации *)
	(* LS01.01-нижн.уровень на входе ОГМ01.04 / защита от сух. хода насоса ФПК *)
	(* ФПК готов к приему осадка *)
	#84 FPKneedToCleanResetFtrig:F_TRIG(CLK: FPKneedToCleanReset)
	#85 FPKstartTrig:RS(SET: pin 1, RESET1: #91)
	out 1 "запуск/старт ФПК" <= #85.Q1
	#86 FPKstopTimer:TOF(IN: pin 1, PT: pin 2)
	#87 FPKstopFtrig:F_TRIG(CLK: #86.Q)
	#88 AND(#85.Q1, #89)
	#89 NOT(pin 11)
	#90 AND(#85.Q1, #92.Q, #94)
	out 2 "ФПК не стартовал" <= #90
	#91 OR(#87.Q, pin 4, pin 5, #93, #95, #98.Q1)
	#92 FPKnotStartedTimer:TON(IN: #88, PT: pin 10)
	#93 NOT(pin 3)
	#94 NOT(pin 9)
	#95 NOT(pin 6)
	#96 AND(#85.Q1, #97)
	#97 GE(pin 7, pin 8)
	#98 FPKneedToCleanTrig:RS(SET: #96, RESET1: #84.Q)
	out 3 "ФПК нужно почистить!" <= #98.Q1
	#99 S FPKneedToCleanReset <= #98.Q1
	#100 FPKneedToCleanResetRtrig:R_TRIG(CLK: pin 6)
	#101 R FPKneedToCleanReset <= #100.Q
END_MACRO
#102 DD1_DO10 <= #83.out 1
#103 FPKnotStarted <= #83.out 2
#104 FPKneedToClean <= #83.out 3
#105 MACRO контроль аналогового входа DD1_AI3(pin 1 "вход": DD1_AI3)
	(* Не смотрим конкретную ошибку, / определяем,что вход неисправен без расшифровки. *)
	#106 DD1_AI3_QE0101:DECODE_FLOAT(VALUE: pin 1, DEF_VALUE: -)
	#107 NE(#106._ERR, 0)
	out 2 "авария" <= #107
	out 1 "выход" <= #106.OUT_VALUE
END_MACRO
#108 DD1_AI3_QE0101value <= #105.out 1
#109 DD1_AI3_error <= #105.out 2
#110 MACRO контроль аналогового входа DD1_AI4(pin 1 "вход": DD1_AI4)
	(* Не смотрим конкретную ошибку, / определяем,что вход неисправен без расшифровки. *)
	#111 DD1_AI4_QE0102:DECODE_FLOAT(VALUE: pin 1, DEF_VALUE: -)
	#112 NE(#111._ERR, 0)
	out 2 "авария" <= #112
	out 1 "выход" <= #111.OUT_VALUE
END_MACRO
#113 DD1_AI4_QE0102value <= #110.out 1
#114 DD1_AI4_error <= #110.out 2
#115 MACRO контроль аналогового входа DD1_AI5(pin 1 "вход": DD1_AI5)
	(* Не смотрим конкретную ошибку, / определяем,что вход неисправен без расшифровки. *)
	#116 DD1_AI5_FPK:DECODE_FLOAT(VALUE: pin 1, DEF_VALUE: -)
	#117 NE(#116._ERR, 0)
	out 2 "авария" <= #117
	out 1 "выход" <= #116.OUT_VALUE
END_MACRO
#118 DD1_AI5_FPKpressureValue <= #115.out 1
#119 DD1_AI5_error <= #115.out 2
#120 MACRO управление НД05.02 УПГ(pin 1 "вход расходомера в куб/час": DD1_AI1_FT0101value, pin 2 "max производительность НД в мл/мин": ND0502setMaxDosVal, pin 3 "задание дозирования в мл/куб": ND0502setKoefProp, pin 4 "режим:1 насос главный": ND0502regimeP1M, pin 5 "режим: 2 насос главный": ND0502regimeP2M, pin 6 "режим: по наработке": ND0502regimeByWT, pin 7 "режим: по кол-ву включений": ND0502regimeByC, pin 8 "авария 1 насоса": DD6_DI.0, pin 9 "авария 2 насоса": DD6_DI.1, pin 10 "сброс аварий": alarmReset, pin 11 "сброс счетчика включений 1 насоса": ND0502resetCountP1, pin 12 "сброс ссчетчика включений 2 насоса": ND0502resetCountP2, pin 13 "сброс наработки 1 насоса": ND0502resetWorkTimeP1, pin 14 "сброс наработки 2 насоса": ND0502resetWorkTimeP2)
	(* Если на входе SEL = TRUE, / то нижнее значение, / иначе - то,что посередине. *)
	(* сигнал 4...20мА на НД05.02/01 *)
	(* сигнал 4...20мА на НД05.02/02 *)
	#121 SEL(#128.pump1ON, 4, #122.outputValue)
	out 6 "выход 4...20мА насоса 1" <= #121
	#122 ND0502dosing:DosingPumpProportional(flowValue: pin 1, setMinPumpDosingValue: -, setMaxPumpDosingValue: pin 2, minOutputValue: -, maxOutputValue: -, setKoeffProportionality: pin 3, minFlowToStart: -)
	out 1 "ошибка блока дозирования" <= #122.dosingError
	#123 SEL(#128.pump2ON, 4, #122.outputValue)
	#124 linTrafND050201:LIN_TRAFO(IN: #123, IN_MIN: 4, IN_MAX: 20, OUT_MIN: 0, OUT_MAX: 1000)
	#125 REAL_TO_WORD(#124.OUT)
	out 7 "выход 4...20мА насоса 2" <= #125
	#126 ND0502regime:choosePumpRegime(start: #122.startDosingPump, pump1Main: pin 4, pump2Main: pin 5, byCounter: #127, byWorkTime: pin 6)
	out 2 "статус: 1 насос главный" <= #126.pump1MainActive
	out 3 "статус: 2 насос главный" <= #126.pump2MainActive
	out 4 "статус: по кол-ву включений" <= #126.byCounterActive
	#127 OR(pin 7, startInitializer)
	out 5 "статус: по наработке" <= #126.byWorkTimeActive
	#128 ND0502manager:TwoPumpManager(startStopPump1: #126.startPump1, startStopPump2: #126.startPump2, alarmPump1: #129, alarmPump2: #130, alarmReset: pin 10, counterStart: #126.startByCounter, Pump1ResetCounter: pin 11, Pump2ResetCounter: pin 12, ValueToResetCounter: -, workTimeStart: #126.startByWorkTime, workTimePump1Reset: pin 13, workTimePump2Reset: pin 14)
	out 12 "сигнал на включение насоса 1" <= #128.pump1ON
	#129 NOT(pin 8)
	out 13 "сигнал на включение насоса 2" <= #128.pump2ON
	out 8 "счетчик включений насоса 1" <= #128.counterPump1
	#130 NOT(pin 9)
	out 9 "счетчик включений насоса 2" <= #128.counterPump2
	out 10 "счетчик наработки насоса 1" <= #128.currentWorkTimePump1
	out 11 "счетчик наработки насоса 2" <= #128.currentWorkTimePump2
END_MACRO
#131 ND0502dosingError <= #120.out 1
#132 ND0502statRegimeP1M <= #120.out 2
#133 ND0502statRegimeP2M <= #120.out 3
#134 ND0502statRegimeByC <= #120.out 4
#135 ND0502statRegimeByWT <= #120.out 5
#136 DD1_AO3 <= #120.out 6
#137 DD10_AO0 <= #120.out 7
#138 ND0502counterP1 <= #120.out 8
#139 ND0502counterP2 <= #120.out 9
#140 ND0502workTimeP1 <= #120.out 10
#141 ND0502workTimeP2 <= #120.out 11
#142 DD4_DO.4 <= #120.out 12
#143 DD4_DO.5 <= #120.out 13
#144 AND(DD2_DO.1, DD5_DI.4)
#145 N0105statStartedP1 <= #144
#146 AND(DD5_DI.4, DD2_DO.2)
#147 N0105statStartedP2 <= #146
#148 MACRO Наполнение РЧВ02.03 (заслонка ЗДЭ02.25)(pin 1 "LS02.02раб.верх.уровень РЧВ": DD6_DI.14, pin 2 "LSA02.01 Перелив РЧВ": DD6_DI.13, pin 3 "статус ЗДЭ02.25 открыт": DD9_DI.0, pin 4 "статус ЗДЭ02.25 закрыт": DD9_DI.1, pin 5 "сброс аварий": alarmReset, pin 6 "время на открытие/закрытие": timeToOpenCloseValve)
	#149 OR(testZDE0225, pin 1)
	#150 NOT(pin 1)
	#151 ZDE0225:SimpleValve(inputOpen: #149, inputClose: #152, statusOpen: pin 3, statusClose: pin 4, reset: pin 5, timeToOpenClose: pin 6)
	out 1 "выход на открытие ЗДЭ02.25" <= #151.outputOpen
	#152 OR(#150, #153)
	out 2 "выход на закрытие ЗДЭ02.25" <= #151.outputClose
	out 3 "авария на открытие ЗДЭ02.25" <= #151.errorToOpen
	#153 NOT(pin 2)
	out 4 "авария на закрытие ЗДЭ02.25" <= #151.errorToClose
END_MACRO
#154 DD4_DO.0 <= #148.out 1
#155 DD4_DO.1 <= #148.out 2
#156 ZDE0225errorToOpen <= #148.out 3
#157 ZDE0225errorToClose <= #148.out 4
#158 MACRO управление Н02.04 (подача из РЧВ)(pin 1 "промывка ФС02.01/01": DD6_DI.20, pin 2 "промывка ФС02.01/02": DD6_DI.22, pin 3 "промывка ФС02.01/03": DD6_DI.24, pin 4 "промывка ФС02.01/04": DD6_DI.26, pin 5 "промывка ФС02.01/05": DD6_DI.28, pin 6 "промывка ФС02.01/06": DD6_DI.30, pin 7 "промывка ФС02.02/01": DD7_DI.0, pin 8 "промывка ФС02.02/02": DD7_DI.2, pin 9 "промывка ФС02.02/03": DD7_DI.4, pin 10 "промывка ФС02.02/04": DD7_DI.6, pin 11 "промывка ФС02.02/05": DD7_DI.8, pin 12 "промывка ФС02.02/06": DD7_DI.10, pin 13 "открыт КЭМ05.01": DD1_DI11, pin 14 "открыт КЭМ06.01": DD1_DI10, pin 15 "открыт КЭМ07.01": DD1_DI9, pin 16 "открыт КЭМ08.01": DD1_DI8, pin 17 "сухой ход Н02.04 (0=сух.ход)": DD5_DI.11, pin 18 "выбрать режим: Н02.04/01 - главный": N0204regimeP1M, pin 19 "выбрать режим: Н02.04/02 - главный": N0204regimeP2M, pin 20 "выбрать режим: по кол-ву включений": N0204regimeByC, pin 21 "выбрать режим: по наработке": N0204regimeWT, pin 22 "авария Н02.04/01 (0=авария)": DD5_DI.7, pin 23 "авария Н02.04/02 (0=авария)": DD5_DI.8, pin 24 "сброс аварий": alarmReset, pin 25 "сброс счетчика включений Н02.04/01": N0204resetCountP1, pin 26 "сброс счетчика включений Н02.04/02": N0204resetCountP2, pin 27 "сброс счетчика наработки Н02.04/01": N0204resetWorkTimeP1, pin 28 "сброс счетчика наработки Н02.04/02": N0204resetWorkTimeP2)
	(* Защита от сухого хода Н02.04 / (LS02.03) 0=сух.ход *)
	(* сброс самоподхвата реле *)
	(* Контроль открытия хотя бы одного из клапанов КЭМ *)
	(* Удержание сигнала на выключение насосов для / гарантированного сброса самоподхвата реле. *)
	(* Проверка, что фильтры 2 / ступени в регенерации (промывке) *)
	(* Проверка, что фильтры 1 / ступени в регенерации (промывке) *)
	#159 OR(pin 1, pin 2, pin 3, pin 4, pin 5, pin 6)
	#160 OR(#159, #161, #162)
	#161 OR(pin 7, pin 8, pin 9, pin 10, pin 11, pin 12)
	#162 OR(pin 13, pin 14, pin 15, pin 16)
	#163 N020401fTrigStop:F_TRIG(CLK: #170.pump1ON)
	#164 AND(#160, pin 17)
	#165 OR(#163.Q, #168.Q)
	#166 N0204stop:TOF(IN: #165, PT: T#1s)
	out 5 "стоп Н02.04" <= #166.Q
	#167 N0204chooseRegime:choosePumpRegime(start: #164, pump1Main: pin 18, pump2Main: pin 19, byCounter: #169, byWorkTime: pin 21)
	out 1 "выбран режим Н02.04/01 = главный" <= #167.pump1MainActive
	#168 N020402fTrigStop:F_TRIG(CLK: #170.pump2ON)
	out 2 "выбран режим Н02.04/02 = главный" <= #167.pump2MainActive
	out 3 "выбран режим по кол-ву включений" <= #167.byCounterActive
	#169 OR(pin 20, startInitializer)
	out 4 "выбран режим по наработке" <= #167.byWorkTimeActive
	#170 N0204manager:TwoPumpManager(startStopPump1: #167.startPump1, startStopPump2: #167.startPump2, alarmPump1: NOT pin 22, alarmPump2: NOT pin 23, alarmReset: pin 24, counterStart: #167.startByCounter, Pump1ResetCounter: pin 25, Pump2ResetCounter: pin 26, ValueToResetCounter: -, workTimeStart: #167.startByWorkTime, workTimePump1Reset: pin 27, workTimePump2Reset: pin 28)
	out 6 "пуск Н02.04/01" <= #170.pump1ON
	out 7 "пуск Н02.04/02" <= #170.pump2ON
	out 8 "счетчик включений Н02.04/01" <= #170.counterPump1
	out 9 "счетчик включений Н02.04/02" <= #170.counterPump2
	out 10 "счетчик наработки Н02.04/01" <= #170.currentWorkTimePump1
	out 11 "счетчик наработки Н02.04/02" <= #170.currentWorkTimePump2
END_MACRO
#171 N0204statRegimeP1M <= #158.out 1
#172 N0204statRegimeP2M <= #158.out 2
#173 N0204statRegimeByC <= #158.out 3
#174 N0204statRegimeWT <= #158.out 4
#175 DD1_DO1 <= #158.out 6
#176 DD1_DO2 <= #158.out 7
#177 N0204counterP1 <= #158.out 8
#178 N0204counterP2 <= #158.out 9
#179 N0204workTimeP1 <= #158.out 10
#180 N0204workTimeP2 <= #158.out 11
#181 OR(panStopN0204, #158.out 5)
#182 DD4_DO.14 <= #181
#183 MACRO управление НД06.02 УПК(pin 1 "вход расходомера в куб/час": DD1_AI2_FT0102value, pin 2 "max производительность НД в мл/мин": ND0602setMaxDosVal, pin 3 "задание дозирования в мл/куб": ND0602setKoefProp, pin 4 "режим:1 насос главный": ND0602regimeP1M, pin 5 "режим: 2 насос главный": ND0602regimeP2M, pin 6 "режим: по наработке": ND0602regimeByWT, pin 7 "режим: по кол-ву включений": ND0602regimeByC, pin 8 "авария 1 насоса": DD6_DI.2, pin 9 "авария 2 насоса": DD6_DI.3, pin 10 "сброс аварий": alarmReset, pin 11 "сброс счетчика включений 1 насоса": ND0602resetCountP1, pin 12 "сброс ссчетчика включений 2 насоса": ND0602resetCountP2, pin 13 "сброс наработки 1 насоса": ND0602resetWorkTimeP1, pin 14 "сброс наработки 2 насоса": ND0602resetWorkTimeP2)
	(* Если на входе SEL = TRUE, / то нижнее значение, / иначе - то,что посередине. *)
	(* сигнал 4...20мА на НД06.02/01 *)
	(* сигнал 4...20мА на НД06.02/02 *)
	#184 SEL(#193.pump1ON, 4, #187.outputValue)
	#185 linTraf060201:LIN_TRAFO(IN: #184, IN_MIN: 4, IN_MAX: 20, OUT_MIN: 0, OUT_MAX: 1000)
	#186 REAL_TO_WORD(#185.OUT)
	out 6 "выход 4...20мА насоса 1" <= #186
	#187 ND0602dosing:DosingPumpProportional(flowValue: pin 1, setMinPumpDosingValue: -, setMaxPumpDosingValue: pin 2, minOutputValue: -, maxOutputValue: -, setKoeffProportionality: pin 3, minFlowToStart: -)
	out 1 "ошибка блока дозирования" <= #187.dosingError
	#188 SEL(#193.pump2ON, 4, #187.outputValue)
	#189 linTraf060202:LIN_TRAFO(IN: #188, IN_MIN: 4, IN_MAX: 20, OUT_MIN: 0, OUT_MAX: 1000)
	#190 REAL_TO_WORD(#189.OUT)
	out 7 "выход 4...20мА насоса 2" <= #190
	#191 ND0602regime:choosePumpRegime(start: #187.startDosingPump, pump1Main: pin 4, pump2Main: pin 5, byCounter: #192, byWorkTime: pin 6)
	out 2 "статус: 1 насос главный" <= #191.pump1MainActive
	out 3 "статус: 2 насос главный" <= #191.pump2MainActive
	out 4 "статус: по кол-ву включений" <= #191.byCounterActive
	#192 OR(pin 7, startInitializer)
	out 5 "статус: по наработке" <= #191.byWorkTimeActive
	#193 ND0602manager:TwoPumpManager(startStopPump1: #191.startPump1, startStopPump2: #191.startPump2, alarmPump1: #194, alarmPump2: #195, alarmReset: pin 10, counterStart: #191.startByCounter, Pump1ResetCounter: pin 11, Pump2ResetCounter: pin 12, ValueToResetCounter: -, workTimeStart: #191.startByWorkTime, workTimePump1Reset: pin 13, workTimePump2Reset: pin 14)
	out 12 "сигнал на включение насоса 1" <= #193.pump1ON
	#194 NOT(pin 8)
	out 13 "сигнал на включение насоса 2" <= #193.pump2ON
	out 8 "счетчик включений насоса 1" <= #193.counterPump1
	#195 NOT(pin 9)
	out 9 "счетчик включений насоса 2" <= #193.counterPump2
	out 10 "счетчик наработки насоса 1" <= #193.currentWorkTimePump1
	out 11 "счетчик наработки насоса 2" <= #193.currentWorkTimePump2
END_MACRO
#196 ND0602dosingError <= #183.out 1
#197 ND0602statRegimeP1M <= #183.out 2
#198 ND0602statRegimeP2M <= #183.out 3
#199 ND0602statRegimeByC <= #183.out 4
#200 ND0602statRegimeByWT <= #183.out 5
#201 DD10_AO1 <= #183.out 6
#202 DD10_AO2 <= #183.out 7
#203 ND0602counterP1 <= #183.out 8
#204 ND0602counterP2 <= #183.out 9
#205 ND0602workTimeP1 <= #183.out 10
#206 ND0602workTimeP2 <= #183.out 11
#207 DD4_DO.6 <= #183.out 12
#208 DD4_DO.7 <= #183.out 13
#209 OR(errorToOpenZDE0301, errorToCloseZDE0301, errorToOpenZDE0302, errorToCloseZDE0302)
#210 OR(DD5_DI.27, #209)
#211 OR(#209, DD5_DI.29)
#212 MACRO Работа УФО03.01(pin 1 "Работа УФО03.01/01": statusUFO030101started, pin 2 "Работа УФО03.01/02": statusUFO030102started, pin 3 "Значение расхода от FT01.02": DD1_AI2_FT0102value, pin 4 "мин.допустимый расход для насосов Н01.05": N0105minFlow, pin 5 "Задержка включения УФО на создание потока": UFO0301startDelayTime, pin 6 "выбор режим: УФО03.01/01 главное": UFO0301regimeP1M, pin 7 "выбор режим: УФО03.01/02 главное": UFO0301regimeP2M, pin 8 "выбор режим: по кол-ву включений": UFO0301regimeByC, pin 9 "выбор режим: по наработке": UFO0301regimeWT, pin 10 "авария УФО03.01/01": #210, pin 11 "авария УФО03.01/02": #211, pin 12 "сброс аварий": alarmReset, pin 13 "сброс счетчика включений УФО03.01/01": UFO0301resetCountP1, pin 14 "сброс счетчика включений УФО03.01/02": UFO0301resetCountP2, pin 15 "сброс счетчика наработки УФО03.01/01": UFO0301resetWorkTimeP1, pin 16 "сброс счетчика наработки УФО03.01/02": UFO0301resetWorkTimeP2)
	(* Включаем УФО, если расходомер показывает расход больше, / чем заданный как минимально допустимый для работы насосов Н01.05. *)
	(* Задержка старта УФО *)
	(* Для подачи предостережения на пульте / оператора (при необходимости), а также / сигнализации лампой АВАРИЯ. *)
	(* Контроль, если УФО включили вручную, / а потока при этом нет. *)
	#213 OR(pin 1, pin 2)
	#214 AND(#213, #215)
	out 1 "УФО вкл без потока" <= #214
	#215 NOT(#217.Q)
	#216 GE(pin 3, pin 4)
	#217 UFO0301startDelay:TON(IN: #216, PT: pin 5)
	#218 UFO0301regimeManager:choosePumpRegime(start: #217.Q, pump1Main: pin 6, pump2Main: pin 7, byCounter: #219, byWorkTime: pin 9)
	out 2 "активен режим - главное УФО 03.01/01" <= #218.pump1MainActive
	out 3 "активен режим - главное УФО 03.01/02" <= #218.pump2MainActive
	out 4 "активен режим - по кол-ву включений" <= #218.byCounterActive
	#219 OR(startInitializer, pin 8)
	out 5 "активен режим - по наработке" <= #218.byWorkTimeActive
	#220 UFO0301manager:TwoPumpManager(startStopPump1: #218.startPump1, startStopPump2: #218.startPump2, alarmPump1: pin 10, alarmPump2: pin 11, alarmReset: pin 12, counterStart: #218.startByCounter, Pump1ResetCounter: pin 13, Pump2ResetCounter: pin 14, ValueToResetCounter: -, workTimeStart: #218.startByWorkTime, workTimePump1Reset: pin 15, workTimePump2Reset: pin 16)
	out 6 "авт. пуск УФО03.01/01" <= #220.pump1ON
	out 7 "авт. пуск УФО03.01/02" <= #220.pump2ON
	out 8 "счетчик включений УФО03.01/01" <= #220.counterPump1
	out 9 "счетчик включений УФО03.01/02" <= #220.counterPump2
	out 10 "счетчик наработки УФО03.01/01" <= #220.currentWorkTimePump1
	out 11 "счетчик наработки УФО03.01/02" <= #220.currentWorkTimePump2
END_MACRO
#221 UFO0301noFlowAttention <= #212.out 1
#222 UFO0301statRegimeP1M <= #212.out 2
#223 UFO0301statRegimeP2M <= #212.out 3
#224 UFO0301statRegimeByC <= #212.out 4
#225 UFO0301statRegimeWT <= #212.out 5
#226 UFO0301counterP1 <= #212.out 8
#227 UFO0301counterP2 <= #212.out 9
#228 UFO0301workTimeP1 <= #212.out 10
#229 UFO0301workTimeP2 <= #212.out 11
#230 MACRO работа задвижек перед УФО и автом.пуск(pin 1 "сигнал на пуск УФО03.01/01": #212.out 6, pin 2 "сигнал на пуск УФО03.01/02": #212.out 7)
	(* 1 = открыть ЗДЭ03.02 / 0 = закрыть ЗДЭ03.02 *)
	(* 1 = открыть ЗДЭ03.01 / 0 = закрыть ЗДЭ03.01 *)
	(* 1 = тест задвижек ЗДЭ / 0 = возможность автом.пуска УФО *)
	(* авт.пускУФО03.01/01 *)
	(* авт.пускУФО03.01/02 *)
	(* авт.стопУФО03.01/01 *)
	(* авт.стопУФО03.01/02 *)
	#231 NOT(testZDE03)
	#232 NOT(testZDE03)
	#233 UFO030101startTrig:R_TRIG(CLK: #235)
	#234 UFO030101start <= #233.Q
	#235 AND(#231, #238, DD1_DI12)
	#236 UFO030101stopTrig:F_TRIG(CLK: #235)
	#237 UFO030101stop <= #236.Q
	#238 SEL(testZDE03, pin 1, manualZDE0301)
	#239 ZDE0301:SimpleValve(inputOpen: #238, inputClose: NOT #238, statusOpen: DD1_DI12, statusClose: DD1_DI13, reset: alarmReset, timeToOpenClose: timeToOpenCloseValve)
	#240 DD4_DO.16 <= #239.outputOpen
	#241 DD4_DO.17 <= #239.outputClose
	#242 errorToOpenZDE0301 <= #239.errorToOpen
	#243 errorToCloseZDE0301 <= #239.errorToClose
	#244 UFO030102startTrig:R_TRIG(CLK: #246)
	#245 UFO030102start <= #244.Q
	#246 AND(#232, #249, DD1_DI14)
	#247 UFO030102stopTrig:F_TRIG(CLK: #246)
	#248 UFO030102stop <= #247.Q
	#249 SEL(testZDE03, pin 2, manualZDE0302)
	#250 ZDE0302:SimpleValve(inputOpen: #249, inputClose: NOT #249, statusOpen: DD1_DI14, statusClose: DD1_DI15, reset: alarmReset, timeToOpenClose: timeToOpenCloseValve)
	#251 DD4_DO.18 <= #250.outputOpen
	#252 DD4_DO.19 <= #250.outputClose
	#253 errorToOpenZDE0302 <= #250.errorToOpen
	#254 errorToCloseZDE0302 <= #250.errorToClose
END_MACRO
#255 MACRO управление НД06.03 УПК(pin 1 "вход расходомера в куб/час": DD1_AI1_FT0101value, pin 2 "max производительность НД в мл/мин": ND0603setMaxDosVal, pin 3 "задание дозирования в мл/куб": ND0603setKoefProp, pin 4 "режим:1 насос главный": ND0603regimeP1M, pin 5 "режим: 2 насос главный": ND0603regimeP2M, pin 6 "режим: по наработке": ND0603regimeByWT, pin 7 "режим: по кол-ву включений": ND0603regimeByC, pin 8 "авария 1 насоса": DD6_DI.4, pin 9 "авария 2 насоса": DD6_DI.5, pin 10 "сброс аварий": alarmReset, pin 11 "сброс счетчика включений 1 насоса": ND0603resetCountP1, pin 12 "сброс ссчетчика включений 2 насоса": ND0603resetCountP2, pin 13 "сброс наработки 1 насоса": ND0603resetWorkTimeP1, pin 14 "сброс наработки 2 насоса": ND0603resetWorkTimeP2)
	(* Если на входе SEL = TRUE, / то нижнее значение, / иначе - то,что посередине. *)
	(* сигнал 4...20мА на НД06.03/01 *)
	(* сигнал 4...20мА на НД06.03/02 *)
	#256 SEL(#265.pump1ON, 4, #259.outputValue)
	#257 linTraf060301:LIN_TRAFO(IN: #256, IN_MIN: 4, IN_MAX: 20, OUT_MIN: 0, OUT_MAX: 1000)
	#258 REAL_TO_WORD(#257.OUT)
	out 6 "выход 4...20мА насоса 1" <= #258
	#259 ND0603dosing:DosingPumpProportional(flowValue: pin 1, setMinPumpDosingValue: -, setMaxPumpDosingValue: pin 2, minOutputValue: -, maxOutputValue: -, setKoeffProportionality: pin 3, minFlowToStart: -)
	out 1 "ошибка блока дозирования" <= #259.dosingError
	#260 SEL(#265.pump2ON, 4, #259.outputValue)
	#261 linTraf060302:LIN_TRAFO(IN: #260, IN_MIN: 4, IN_MAX: 20, OUT_MIN: 0, OUT_MAX: 1000)
	#262 REAL_TO_WORD(#261.OUT)
	out 7 "выход 4...20мА насоса 2" <= #262
	#263 ND0603regime:choosePumpRegime(start: #259.startDosingPump, pump1Main: pin 4, pump2Main: pin 5, byCounter: #264, byWorkTime: pin 6)
	out 2 "статус: 1 насос главный" <= #263.pump1MainActive
	out 3 "статус: 2 насос главный" <= #263.pump2MainActive
	out 4 "статус: по кол-ву включений" <= #263.byCounterActive
	#264 OR(pin 7, startInitializer)
	out 5 "статус: по наработке" <= #263.byWorkTimeActive
	#265 ND0603manager:TwoPumpManager(startStopPump1: #263.startPump1, startStopPump2: #263.startPump2, alarmPump1: #266, alarmPump2: #267, alarmReset: pin 10, counterStart: #263.startByCounter, Pump1ResetCounter: pin 11, Pump2ResetCounter: pin 12, ValueToResetCounter: -, workTimeStart: #263.startByWorkTime, workTimePump1Reset: pin 13, workTimePump2Reset: pin 14)
	out 12 "сигнал на включение насоса 1" <= #265.pump1ON
	#266 NOT(pin 8)
	out 13 "сигнал на включение насоса 2" <= #265.pump2ON
	out 8 "счетчик включений насоса 1" <= #265.counterPump1
	#267 NOT(pin 9)
	out 9 "счетчик включений насоса 2" <= #265.counterPump2
	out 10 "счетчик наработки насоса 1" <= #265.currentWorkTimePump1
	out 11 "счетчик наработки насоса 2" <= #265.currentWorkTimePump2
END_MACRO
#268 ND0603dosingError <= #255.out 1
#269 ND0603statRegimeP1M <= #255.out 2
#270 ND0603statRegimeP2M <= #255.out 3
#271 ND0603statRegimeByC <= #255.out 4
#272 ND0603statRegimeByWT <= #255.out 5
#273 DD10_AO3 <= #255.out 6
#274 DD10_AO4 <= #255.out 7
#275 ND0603counterP1 <= #255.out 8
#276 ND0603counterP2 <= #255.out 9
#277 ND0603workTimeP1 <= #255.out 10
#278 ND0603workTimeP2 <= #255.out 11
#279 DD4_DO.8 <= #255.out 12
#280 DD4_DO.9 <= #255.out 13
#281 MACRO управление Н04.04 (дренажные)(pin 1 "защита от сухого хода Н04.04": DD5_DI.18, pin 2 "автоматич.пускН04.04": DD5_DI.19, pin 3 "режим Н04.04/01 главный": N0404regimeP1M, pin 4 "режим Н04.04/02 главный": N0404regimeP2M, pin 5 "режим по кол-ву включений": N0404regimeByC, pin 6 "режим по наработке": N0404regimeWT, pin 7 "авария Н04.04/01": DD5_DI.15, pin 8 "авария Н04.04/02": DD5_DI.14, pin 9 "сброс аварий": alarmReset, pin 10 "сброс счетчика включений Н04.04/01": N0404resetCountP1, pin 11 "сброс счетчика включений Н04.04/02": N0404resetCountP2, pin 12 "сброс счетчика наработки Н04.04/01": N0404resetWorkTimeP1, pin 13 "сброс счетчика наработки Н04.04/02": N0404resetWorkTimeP2)
	(* 0=авария *)
	(* сухой ход Н04.04 / 0=защита *)
	(* от поплавка *)
	(* насосы имеют электрическую блокировку / от одновременного включения *)
	(* Излишняя перестраховка по сухому ходу, / на уровне реле уже все отрабатывается. *)
	(* сбрасывает самоподхват пускового реле *)
	#282 NOT(pin 1)
	out 1 "стоп Н04.04" <= #282
	#283 AND(pin 1, pin 2)
	#284 N0401choosePumpRegime:choosePumpRegime(start: #283, pump1Main: pin 3, pump2Main: pin 4, byCounter: #285, byWorkTime: pin 6)
	out 2 "выбран режим: Н04.04/01 главный" <= #284.pump1MainActive
	out 3 "выбран режим: Н04.04/02 главный" <= #284.pump2MainActive
	out 4 "выбран режим: по кол-ву включений" <= #284.byCounterActive
	#285 OR(startInitializer, pin 5)
	out 5 "выбран режим: по наработке" <= #284.byWorkTimeActive
	#286 N0404twoPumpManager:TwoPumpManager(startStopPump1: #284.startPump1, startStopPump2: #284.startPump2, alarmPump1: #287, alarmPump2: #288, alarmReset: pin 9, counterStart: #284.startByCounter, Pump1ResetCounter: pin 10, Pump2ResetCounter: pin 11, ValueToResetCounter: -, workTimeStart: #284.startByWorkTime, workTimePump1Reset: pin 12, workTimePump2Reset: pin 13)
	out 6 "пуск Н04.04/01" <= #286.pump1ON
	#287 NOT(pin 7)
	out 7 "пуск Н04.04/02" <= #286.pump2ON
	out 8 "счетчик кол-ва включений Н04.04/01" <= #286.counterPump1
	#288 NOT(pin 8)
	out 9 "счетчик кол-ва включений Н04.04/02" <= #286.counterPump2
	out 10 "счетчик времени наработки Н04.04/01" <= #286.currentWorkTimePump1
	out 11 "счетчик времени наработки Н04.04/02" <= #286.currentWorkTimePump2
END_MACRO
#289 DD4_DO.15 <= #281.out 1
#290 N0404statRegimeP1M <= #281.out 2
#291 N0404statRegimeP2M <= #281.out 3
#292 N0404statRegimeByC <= #281.out 4
#293 N0404statRegimeWT <= #281.out 5
#294 DD1_DO5 <= #281.out 6
#295 DD1_DO6 <= #281.out 7
#296 N0404counterP1 <= #281.out 8
#297 N0404counterP2 <= #281.out 9
#298 N0404workTimeP1 <= #281.out 10
#299 N0404workTimeP2 <= #281.out 11
#300 MACRO управление НД07.03 УПЩ (поддержка рН, ПИД-регулятор)(pin 1 "вход рН-метра QE01.01": DD1_AI3_QE0101value, pin 2 "уставка рН": ND0703pHsetValue, pin 3 "режим:1 насос главный": ND0703regimeP1M, pin 4 "режим: 2 насос главный": ND0703regimeP2M, pin 5 "режим: по наработке": ND0703regimeByWT, pin 6 "режим: по кол-ву включений": ND0703regimeByC, pin 7 "авария 1 насоса": DD6_DI.6, pin 8 "авария 2 насоса": DD6_DI.7, pin 9 "сброс аварий": alarmReset, pin 10 "сброс счетчика включений 1 насоса": ND0703resetCountP1, pin 11 "сброс счетчика включений 2 насоса": ND0703resetCountP2, pin 12 "сброс наработки 1 насоса": ND0703resetWorkTimeP1, pin 13 "сброс наработки 2 насоса": ND0703resetWorkTimeP2, pin 14 "ручное управл.выходом Y (4...20мА)": ND0703YoutManual, pin 15 "1=ручное/0=автомат.управл.": ND0703YmanAuto, pin 16 "вход расходомера FT01.01 (куб.м/час)": DD1_AI1_FT0101value, pin 17 "коэфф.I": ND0703koeffI, pin 18 "коэфф.D": ND0703koeffD, pin 19 "коэфф.Р": ND0703koeffP)
	(* min расход в кубометрах в час / для неачала дозирования. *)
	(* Если на входе SEL = TRUE, / то нижнее значение, / иначе - то,что посередине. *)
	(* сигнал 4...20мА на НД07.03/01 *)
	(* сигнал 4...20мА на НД07.03/02 *)
	#301 ND0703pidReg:PID(ACTUAL: pin 1, SET_POINT: pin 2, KP: pin 19, TN: pin 17, TV: pin 18, Y_MANUAL: pin 14, Y_OFFSET: 12, Y_MIN: 0, Y_MAX: 1000, MANUAL: pin 15, RESET: #301.OVERFLOW)
	#302 SEL(#309.pump1ON, 0, #301.Y)
	#303 REAL_TO_WORD(#302)
	out 5 "выход 4...20мА насоса 1" <= #303
	#304 SEL(#309.pump2ON, 0, #301.Y)
	#305 REAL_TO_WORD(#304)
	out 6 "выход 4...20мА насоса 2" <= #305
	#306 GE(pin 16, 10)
	#307 ND0703regime:choosePumpRegime(start: #306, pump1Main: pin 3, pump2Main: pin 4, byCounter: #308, byWorkTime: pin 5)
	out 1 "статус: 1 насос главный" <= #307.pump1MainActive
	out 2 "статус: 2 насос главный" <= #307.pump2MainActive
	out 3 "статус: по кол-ву включений" <= #307.byCounterActive
	out 4 "статус: по наработке" <= #307.byWorkTimeActive
	#308 OR(pin 6, startInitializer)
	#309 ND0703manager:TwoPumpManager(startStopPump1: #307.startPump1, startStopPump2: #307.startPump2, alarmPump1: #310, alarmPump2: #311, alarmReset: pin 9, counterStart: #307.startByCounter, Pump1ResetCounter: pin 10, Pump2ResetCounter: pin 11, ValueToResetCounter: -, workTimeStart: #307.startByWorkTime, workTimePump1Reset: pin 12, workTimePump2Reset: pin 13)
	out 11 "сигнал на включение насоса 1" <= #309.pump1ON
	#310 NOT(pin 7)
	out 12 "сигнал на включение насоса 2" <= #309.pump2ON
	out 7 "счетчик включений насоса 1" <= #309.counterPump1
	#311 NOT(pin 8)
	out 8 "счетчик включений насоса 2" <= #309.counterPump2
	out 9 "счетчик наработки насоса 1" <= #309.currentWorkTimePump1
	out 10 "счетчик наработки насоса 2" <= #309.currentWorkTimePump2
END_MACRO
#312 ND0703statRegimeP1M <= #300.out 1
#313 ND0703statRegimeP2M <= #300.out 2
#314 ND0703statRegimeByC <= #300.out 3
#315 ND0703statRegimeByWT <= #300.out 4
#316 DD10_AO5 <= #300.out 5
#317 DD10_AO6 <= #300.out 6
#318 ND0703counterP1 <= #300.out 7
#319 ND0703counterP2 <= #300.out 8
#320 ND0703workTimeP1 <= #300.out 9
#321 ND0703workTimeP2 <= #300.out 10
#322 DD4_DO.10 <= #300.out 11
#323 DD4_DO.11 <= #300.out 12
#324 MACRO импульсный счетчик FQS0301(pin 1 "вход от счетчика": DD6_DI.19, pin 2 "вес импульса счетчика": FQS0301impulsValue, pin 3 "сброс счетчика": FQS0301reset, pin 4 "величина коррекции счетчика": FQS0301correction, pin 5 "прибавить коррекцию": FQS0301addCorrection, pin 6 "вычесть коррекцию": FQS0301deleteCorrection)
	(* число, коорое будем прибавлять или / вычитать из накопленной суммы стоков. *)
	(* коррекция показаний счетчика. *)
	(* Если в результате коррекции накопленная сумма станет меньше нуля, то она принудительно станет равна нулю. *)
	(* значение в REAL (в какой-то момент начинает / отображаться в экспоненциальной форме) *)
	(* сброс показаний счетчика *)
	#325 FQS0301rTrig:R_TRIG(CLK: pin 1)
	#326 ADD(EN: #325.Q, FQS0301totalAmount, pin 2)
	out 1 "накопленная сумма стоков (REAL)" <= #326
	#327 FQS0301resetRtrig:R_TRIG(CLK: pin 3)
	#328 MOVE(EN: #327.Q, 0)
	#329 FQS0301totalAmount <= #328
	#330 FQS0301addCorrRtrig:R_TRIG(CLK: pin 5)
	#331 ADD(EN: #330.Q, FQS0301totalAmount, pin 4)
	#332 FQS0301totalAmount <= #331
	#333 FQS0301deleteCorrRtrig:R_TRIG(CLK: pin 6)
	#334 SUB(EN: #333.Q, FQS0301totalAmount, pin 4)
	#335 FQS0301totalAmount <= #334
	#336 LT(FQS0301totalAmount, 0)
	#337 MOVE(EN: #336, 0)
	#338 FQS0301totalAmount <= #337
END_MACRO
#339 FQS0301totalAmount <= #324.out 1
#340 MACRO управление НД08.03 УПФ(pin 1 "вход расходомера в куб/час": DD1_AI1_FT0101value, pin 2 "max производительность НД в мл/мин": ND0803setMaxDosVal, pin 3 "задание дозирования в мл/куб": ND0803setKoefProp, pin 4 "режим:1 насос главный": ND0803regimeP1M, pin 5 "режим: 2 насос главный": ND0803regimeP2M, pin 6 "режим: по наработке": ND0803regimeByWT, pin 7 "режим: по кол-ву включений": ND0803regimeByC, pin 8 "авария 1 насоса": DD5_DI.12, pin 9 "авария 2 насоса": DD5_DI.13, pin 10 "сброс аварий": alarmReset, pin 11 "сброс счетчика включений 1 насоса": ND0803resetCountP1, pin 12 "сброс ссчетчика включений 2 насоса": ND0803resetCountP2, pin 13 "сброс наработки 1 насоса": ND0803resetWorkTimeP1, pin 14 "сброс наработки 2 насоса": ND0803resetWorkTimeP2, pin 15 "сухой ход 1 насоса": DD1_DI6, pin 16 "сухой ход 2 насоса": DD1_DI7)
	(* Если на входе SEL = TRUE, / то нижнее значение, / иначе - то,что посередине. *)
	(* сигнал 4...20мА на НД08.03/01 *)
	(* сигнал 4...20мА на НД08.03/02 *)
	#341 SEL(#350.pump1ON, 0, #342.outputValue)
	out 6 "выход 4...20мА насоса 1" <= #341
	#342 ND0803dosing:DosingPumpProportional(flowValue: pin 1, setMinPumpDosingValue: -, setMaxPumpDosingValue: pin 2, minOutputValue: -, maxOutputValue: -, setKoeffProportionality: pin 3, minFlowToStart: -)
	out 1 "ошибка блока дозирования" <= #342.dosingError
	#343 SEL(#350.pump2ON, 0, #342.outputValue)
	out 7 "выход 4...20мА насоса 2" <= #343
	#344 ND0803regime:choosePumpRegime(start: #342.startDosingPump, pump1Main: pin 4, pump2Main: pin 5, byCounter: #345, byWorkTime: pin 6)
	out 2 "статус: 1 насос главный" <= #344.pump1MainActive
	out 3 "статус: 2 насос главный" <= #344.pump2MainActive
	out 4 "статус: по кол-ву включений" <= #344.byCounterActive
	#345 OR(pin 7, startInitializer)
	out 5 "статус: по наработке" <= #344.byWorkTimeActive
	out 12 "сигнал на включение насоса 1" <= #350.pump1ON
	#346 NOT(pin 8)
	#347 OR(#346, pin 15)
	out 13 "сигнал на включение насоса 2" <= #350.pump2ON
	#348 NOT(pin 9)
	#349 OR(#348, pin 16)
	#350 ND0803manager:TwoPumpManager(startStopPump1: #344.startPump1, startStopPump2: #344.startPump2, alarmPump1: #347, alarmPump2: #349, alarmReset: pin 10, counterStart: #344.startByCounter, Pump1ResetCounter: pin 11, Pump2ResetCounter: pin 12, ValueToResetCounter: -, workTimeStart: #344.startByWorkTime, workTimePump1Reset: pin 13, workTimePump2Reset: pin 14)
	out 8 "счетчик включений насоса 1" <= #350.counterPump1
	out 9 "счетчик включений насоса 2" <= #350.counterPump2
	out 10 "счетчик наработки насоса 1" <= #350.currentWorkTimePump1
	out 11 "счетчик наработки насоса 2" <= #350.currentWorkTimePump2
END_MACRO
#351 ND0803dosingError <= #340.out 1
#352 ND0803statRegimeP1M <= #340.out 2
#353 ND0803statRegimeP2M <= #340.out 3
#354 ND0803statRegimeByC <= #340.out 4
#355 ND0803statRegimeByWT <= #340.out 5
#356 DD1_AO1 <= #340.out 6
#357 DD1_AO2 <= #340.out 7
#358 ND0803counterP1 <= #340.out 8
#359 ND0803counterP2 <= #340.out 9
#360 ND0803workTimeP1 <= #340.out 10
#361 ND0803workTimeP2 <= #340.out 11
#362 DD1_DO3 <= #340.out 12
#363 DD1_DO4 <= #340.out 13
#364 AND(DD1_DI5, DD1_DI4, DD6_DI.11)
#365 DD1_DO8 <= #364
#366 EQ(lastError, 0)
#367 alarmPLKnetworkDelay:TOF(IN: #366, PT: T#20s)
#368 NOT(#367.Q)
#369 alarmPLKnetwork <= #368
#370 MACRO управление НД08.04 УПФ(pin 1 "насос Н04.01 работает": DD7_DI.13, pin 2 "авария НД08.04": DD6_DI.16, pin 3 "уставкаНД08.04(0...100%)": ND0804doseValue)
	(* Преобразует сигнал 0...100 / пропорционально в 4...20мА *)
	#371 AND(pin 1, pin 2)
	out 1 "пуск/стоп НД08.04" <= #371
	#372 ND0804linearTransformator:LIN_TRAFO(IN: pin 3, IN_MIN: 0, IN_MAX: 100, OUT_MIN: 0, OUT_MAX: 1000)
	#373 REAL_TO_WORD(#372.OUT)
	out 2 "управление НД08.04 (4...20мА)" <= #373
	out 3 "ошибка блока дозирования" <= #372.ERROR
END_MACRO
#374 DD4_DO.12 <= #370.out 1
#375 DD10_AO7 <= #370.out 2
#376 ND0804dosingError <= #370.out 3
#377 NOT(DD6_DI.0)
#378 alarmND050201 <= #377
#379 NOT(DD6_DI.23)
#380 alarmFS020102 <= #379
#381 NOT(DD9_DI.14)
#382 alarmZDE0211power <= #381
#383 NOT(DD6_DI.1)
#384 alarmND050202 <= #383
#385 NOT(DD6_DI.25)
#386 alarmFS020103 <= #385
#387 NOT(DD9_DI.15)
#388 alarmZDE0212power <= #387
#389 NOT(DD6_DI.2)
#390 alarmND060201 <= #389
#391 NOT(DD6_DI.27)
#392 alarmFS020104 <= #391
#393 NOT(DD9_DI.16)
#394 alarmZDE0213power <= #393
#395 NOT(DD6_DI.3)
#396 alarmND060202 <= #395
#397 NOT(DD6_DI.29)
#398 alarmFS020105 <= #397
#399 NOT(DD9_DI.17)
#400 alarmZDE0214power <= #399
#401 MACRO контроль включения мешалок(pin 1 "работа НД06.02/01": DD4_DO.6, pin 2 "работа НД06.02/02": DD4_DO.7, pin 3 "работа НД06.03/01": DD4_DO.8, pin 4 "работа НД06.03/02": DD4_DO.9, pin 5 "работа мешалки М06.04": DD5_DI.21, pin 6 "работа НД07.03/01": DD4_DO.10, pin 7 "работа НД07.03/02": DD4_DO.11, pin 8 "работа мешалки М07.02": DD5_DI.23, pin 9 "работа НД08.03/01": DD1_DO3, pin 10 "работа НД08.03/02": DD1_DO4, pin 11 "работа НД08.04": DD4_DO.12, pin 12 "работа мешалки М08.02": DD5_DI.25)
	#402 OR(pin 1, pin 2, pin 3, pin 4)
	#403 AND(#402, #404)
	out 1 "дозирования при выключенной М06.04" <= #403
	#404 NOT(pin 5)
	#405 OR(pin 6, pin 7)
	#406 AND(#405, #407)
	out 2 "дозирования при выключенной М07.02" <= #406
	#407 NOT(pin 8)
	#408 OR(pin 9, pin 10, pin 11)
	#409 AND(#408, #410)
	out 3 "дозирования при выключенной М08.02" <= #409
	#410 NOT(pin 12)
END_MACRO
#411 M0604attention <= #401.out 1
#412 M0702attention <= #401.out 2
#413 M0802attention <= #401.out 3
#414 NOT(DD6_DI.4)
#415 alarmND060301 <= #414
#416 NOT(DD6_DI.31)
#417 alarmFS020106 <= #416
#418 NOT(DD9_DI.18)
#419 alarmZDE0215power <= #418
#420 NOT(DD6_DI.5)
#421 alarmND060302 <= #420
#422 NOT(DD7_DI.1)
#423 alarmFS020201 <= #422
#424 NOT(DD9_DI.19)
#425 alarmZDE0216power <= #424
#426 NOT(DD6_DI.6)
#427 alarmND070301 <= #426
#428 NOT(DD7_DI.3)
#429 alarmFS020202 <= #428
#430 NOT(DD9_DI.20)
#431 alarmZDE0217power <= #430
#432 NOT(DD6_DI.7)
#433 alarmND070302 <= #432
#434 NOT(DD7_DI.5)
#435 alarmFS020203 <= #434
#436 NOT(DD9_DI.21)
#437 alarmZDE0218power <= #436
#438 NOT(DD5_DI.12)
#439 alarmND080301 <= #438
#440 NOT(DD7_DI.7)
#441 alarmFS020204 <= #440
#442 NOT(DD9_DI.22)
#443 alarmZDE0219power <= #442
#444 NOT(DD5_DI.13)
#445 alarmND080302 <= #444
#446 NOT(DD7_DI.9)
#447 alarmFS020205 <= #446
#448 NOT(DD9_DI.23)
#449 alarmZDE0220power <= #448
#450 NOT(DD6_DI.16)
#451 alarmND0804 <= #450
#452 NOT(DD7_DI.11)
#453 alarmFS020206 <= #452
#454 NOT(DD9_DI.24)
#455 alarmZDE0221power <= #454
#456 NOT(DD6_DI.11)
#457 alarmOGM0104overload <= #456
#458 NOT(DD9_DI.4)
#459 alarmZDE0201power <= #458
#460 NOT(DD9_DI.25)
#461 alarmZDE0222power <= #460
#462 MACRO переменные для обмена с панелью()
	#463 MACRO PSW регистры на передачу в панель (отображение)()
		(* panFQS0301totalAmount - переменная отображена сразу на выходе соответствующего макроса (учет очищенных стоков). / Здесь не хранится. *)
		(* PSW регистры на передачу в панель (отображение) *)
		#464 panFT0101value <= DD1_AI1_FT0101value
		#465 panQE0101value <= DD1_AI3_QE0101value
		#466 panFT0102value <= DD1_AI2_FT0102value
		#467 panQE0102value <= DD1_AI4_QE0102value
		#468 panFPKpressureValue <= DD1_AI5_FPKpressureValue
		#469 panFQS0301total <= FQS0301totalAmount
		#470 panTemperature <= temperatureValue
		#471 MACRO Время наработки и кол-во включений агрегатов()
			#472 workTimeND050201:TimeFromWorkTime(input: ND0502workTimeP1)
			#473 panND050201workDays <= #472.days
			#474 panND050201workHours <= #472.hours
			#475 panND050201workMinutes <= #472.minutes
			#476 panND050201workSeconds <= #472.seconds
			#477 workTimeND050202:TimeFromWorkTime(input: ND0502workTimeP2)
			#478 panND050202workDays <= #477.days
			#479 panND050202workHours <= #477.hours
			#480 panND050202workMinutes <= #477.minutes
			#481 panND050202workSeconds <= #477.seconds
			#482 panND0502counterP1 <= ND0502counterP1
			#483 panND0502counterP2 <= ND0502counterP2
			#484 workTimeND060201:TimeFromWorkTime(input: ND0602workTimeP1)
			#485 panND060201workDays <= #484.days
			#486 panND060201workHours <= #484.hours
			#487 panND060201workMinutes <= #484.minutes
			#488 panND060201workSeconds <= #484.seconds
			#489 workTimeND060202:TimeFromWorkTime(input: ND0602workTimeP2)
			#490 panND060202workDays <= #489.days
			#491 panND060202workHours <= #489.hours
			#492 panND060202workMinutes <= #489.minutes
			#493 panND060202workSeconds <= #489.seconds
			#494 panND0602counterP1 <= ND0602counterP1
			#495 panND0602counterP2 <= ND0602counterP2
			#496 workTimeND060301:TimeFromWorkTime(input: ND0603workTimeP1)
			#497 panND060301workDays <= #496.days
			#498 panND060301workHours <= #496.hours
			#499 panND060301workMinutes <= #496.minutes
			#500 panND060301workSeconds <= #496.seconds
			#501 workTimeND060302:TimeFromWorkTime(input: ND0603workTimeP2)
			#502 panND060302workDays <= #501.days
			#503 panND060302workHours <= #501.hours
			#504 panND060302workMinutes <= #501.minutes
			#505 panND060302workSeconds <= #501.seconds
			#506 panND0603counterP1 <= ND0603counterP1
			#507 panND0603counterP2 <= ND0603counterP2
			#508 workTimeND070301:TimeFromWorkTime(input: ND0703workTimeP1)
			#509 panND070301workDays <= #508.days
			#510 panND070301workHours <= #508.hours
			#511 panND070301workMinutes <= #508.minutes
			#512 panND070301workSeconds <= #508.seconds
			#513 workTimeND070302:TimeFromWorkTime(input: ND0703workTimeP2)
			#514 panND070302workDays <= #513.days
			#515 panND070302workHours <= #513.hours
			#516 panND070302workMinutes <= #513.minutes
			#517 panND070302workSeconds <= #513.seconds
			#518 panND0703counterP1 <= ND0703counterP1
			#519 panND0703counterP2 <= ND0703counterP2
			#520 workTimeND080301:TimeFromWorkTime(input: ND0803workTimeP1)
			#521 panND080301workDays <= #520.days
			#522 panND080301workHours <= #520.hours
			#523 panND080301workMinutes <= #520.minutes
			#524 panND080301workSeconds <= #520.seconds
			#525 workTimeND080302:TimeFromWorkTime(input: ND0803workTimeP2)
			#526 panND080302workDays <= #525.days
			#527 panND080302workHours <= #525.hours
			#528 panND080302workMinutes <= #525.minutes
			#529 panND080302workSeconds <= #525.seconds
			#530 panND0803counterP1 <= ND0803counterP1
			#531 panND0803counterP2 <= ND0803counterP2
			#532 workTimeN010501:TimeFromWorkTime(input: N0105workTimeP1)
			#533 panN010501workDays <= #532.days
			#534 panN010501workHours <= #532.hours
			#535 panN010501workMinutes <= #532.minutes
			#536 panN010501workSeconds <= #532.seconds
			#537 workTimeN010502:TimeFromWorkTime(input: N0105workTimeP2)
			#538 panN010502workDays <= #537.days
			#539 panN010502workHours <= #537.hours
			#540 panN010502workMinutes <= #537.minutes
			#541 panN010502workSeconds <= #537.seconds
			#542 panN0105counterP1 <= N0105counterP1
			#543 panN0105counterP2 <= N0105counterP2
			#544 workTimeN020401:TimeFromWorkTime(input: N0204workTimeP1)
			#545 panN020401workDays <= #544.days
			#546 panN020401workHours <= #544.hours
			#547 panN020401workMinutes <= #544.minutes
			#548 panN020401workSeconds <= #544.seconds
			#549 workTimeN020402:TimeFromWorkTime(input: N0204workTimeP2)
			#550 panN020402workDays <= #549.days
			#551 panN020402workHours <= #549.hours
			#552 panN020402workMinutes <= #549.minutes
			#553 panN020402workSeconds <= #549.seconds
			#554 panN0204counterP1 <= N0204counterP1
			#555 panN0204counterP2 <= N0204counterP2
			#556 workTimeN040401:TimeFromWorkTime(input: N0404workTimeP1)
			#557 panN040401workDays <= #556.days
			#558 panN040401workHours <= #556.hours
			#559 panN040401workMinutes <= #556.minutes
			#560 panN040401workSeconds <= #556.seconds
			#561 workTimeN040402:TimeFromWorkTime(input: N0404workTimeP2)
			#562 panN040402workDays <= #561.days
			#563 panN040402workHours <= #561.hours
			#564 panN040402workMinutes <= #561.minutes
			#565 panN040402workSeconds <= #561.seconds
			#566 panN0404counterP1 <= N0404counterP1
			#567 panN0404counterP2 <= N0404counterP2
			#568 workTimeUFO030101:TimeFromWorkTime(input: UFO0301workTimeP1)
			#569 panUFO030101workDays <= #568.days
			#570 panUFO030101workHours <= #568.hours
			#571 panUFO030101workMinutes <= #568.minutes
			#572 panUFO030101workSeconds <= #568.seconds
			#573 workTimeUFO030102:TimeFromWorkTime(input: UFO0301workTimeP2)
			#574 panUFO030102workDays <= #573.days
			#575 panUFO030102workHours <= #573.hours
			#576 panUFO030102workMinutes <= #573.minutes
			#577 panUFO030102workSeconds <= #573.seconds
			#578 panUFO0301counterP1 <= UFO0301counterP1
			#579 panUFO0301counterP2 <= UFO0301counterP2
		END_MACRO
		#580 panVolumeToRegen <= volumeToRegen
	END_MACRO
	#581 MACRO PSB регистры на передачу в панель (отображение)()
		(* PSB регистры на передачу в панель (отображение) *)
		#582 MACRO 8 bit output module 1()
			#583 panStartND050201 <= DD4_DO.4
			#584 panStartND050202 <= DD4_DO.5
			#585 panStartND060201 <= DD4_DO.6
			#586 panStartND060202 <= DD4_DO.7
			#587 panStartND060301 <= DD4_DO.8
			#588 panStartND060302 <= DD4_DO.9
			#589 panStartM0604 <= DD5_DI.21
			#590 panStartND070301 <= DD4_DO.10
		END_MACRO
		#591 MACRO 8 bit output module 2()
			#592 panStartND070302 <= DD4_DO.11
			#593 panStartM0702 <= DD5_DI.23
			#594 panStartND080301 <= DD1_DO3
			#595 panStartND080302 <= DD1_DO4
			#596 panStartND0804 <= DD4_DO.12
			#597 panStartM0802 <= DD5_DI.25
			#598 panStartN020401 <= DD5_DI.9
			#599 panStartN020402 <= DD5_DI.10
		END_MACRO
		#600 MACRO 8 bit output module 3()
			#601 panStartN010501 <= N0105statStartedP1
			#602 panStartN010502 <= N0105statStartedP2
			#603 panCleanFS020101 <= DD6_DI.20
			#604 panCleanFS020102 <= DD6_DI.22
			#605 panCleanFS020103 <= DD6_DI.24
			#606 panCleanFS020104 <= DD6_DI.26
			#607 panCleanFS020105 <= DD6_DI.28
			#608 panCleanFS020106 <= DD6_DI.30
		END_MACRO
		#609 MACRO 8 bit output module 4()
			#610 panCleanFS020201 <= DD7_DI. 0
			#611 panCleanFS020202 <= DD7_DI. 2
			#612 panCleanFS020203 <= DD7_DI. 4
			#613 panCleanFS020204 <= DD7_DI. 6
			#614 panCleanFS020205 <= DD7_DI. 8
			#615 panCleanFS020206 <= DD7_DI. 10
			#616 panSludgeReady <= DD7_DI.15
			#617 panStartN0401 <= DD7_DI.13
		END_MACRO
		#618 MACRO 8 bit output module 5()
			#619 panKSHE0401open <= DD9_DI.2
			#620 panFPKready <= DD7_DI.12
			#621 panFPKneedToClean <= FPKneedToClean
			#622 panStartN040401 <= DD5_DI.16
			#623 panStartN040402 <= DD5_DI.17
			#624 panStartUFO030101 <= statusUFO030101started
			#625 panStartUFO030102 <= statusUFO030102started
			#626 panAlarm <= alarm
		END_MACRO
		#627 MACRO 8 bit output module 6()
			#628 panErrorTempSensor <= DD1_AI0_error
			#629 panErrorFT0101 <= DD1_AI1_error
			#630 panErrorFT0102 <= DD1_AI2_error
			#631 panErrorQE0102 <= DD1_AI3_error
			#632 panErrorQE0102 <= DD1_AI4_error
			#633 panAlarmHighTemp <= alarmHighTemperature
			#634 panAlarmLowTemp <= alarmLowTemperature
			#635 panND0502dosingError <= ND0502dosingError
		END_MACRO
		#636 MACRO 8 bit output module 7()
			#637 panND0602dosingError <= ND0602dosingError
			#638 panND0603dosingError <= ND0603dosingError
			#639 panND0803dosingError <= ND0803dosingError
			#640 panND0804dosingError <= ND0804dosingError
			#641 panND080301emptyAlarm <= DD1_DI6
			#642 panND080302emptyAlarm <= DD1_DI7
			#643 panN010501alarm <= N010501alarm
			#644 panN010502alarm <= N010502alarm
		END_MACRO
		#645 MACRO 8 bit output module 8()
			#646 panZDE0225errorToOpen <= ZDE0225errorToOpen
			#647 panZDE0225errorToClose <= ZDE0225errorToClose
			#648 panFPKalarm <= DD7_DI.14
			#649 panFPKnotStarted <= FPKnotStarted
			#650 panErrorFPKsensor <= DD1_AI5_error
			#651 panFPKkshe0401errorToOpen <= FPKkshe0401errorToOpen
			#652 panFPKkshe0401errorToClose <= FPKkshe0401errorToClose
			#653 panUFO030101alarm <= statusUFO030101alarm
		END_MACRO
		#654 MACRO 8 bit output module 9()
			#655 panUFO030102alarm <= statusUFO030102alarm
			#656 panFilterFailToRegen020101 <= filterFailToRegen020101
			#657 panErrorToOpenZD0201 <= errorToOpenZD0201
			#658 panErrorToCloseZD0201 <= errorToCloseZD0201
			#659 panErrorToOpenZD0207 <= errorToOpenZD0207
			#660 panErrorToCloseZD0207 <= errorToCloseZD0207
			#661 panFilterFailToRegen020102 <= filterFailToRegen020102
			#662 panErrorToOpenZD0202 <= errorToOpenZD0202
		END_MACRO
		#663 MACRO 8 bit output module 10()
			#664 panErrorToCloseZD0202 <= errorToCloseZD0202
			#665 panErrorToOpenZD0208 <= errorToOpenZD0208
			#666 panErrorToCloseZD0208 <= errorToCloseZD0208
			#667 panFilterFailToRegen020103 <= filterFailToRegen020103
			#668 panErrorToOpenZD0203 <= errorToOpenZD0203
			#669 panErrorToCloseZD0203 <= errorToCloseZD0203
			#670 panErrorToOpenZD0209 <= errorToOpenZD0209
			#671 panErrorToCloseZD0209 <= errorToCloseZD0209
		END_MACRO
		#672 MACRO 8 bit output module 11()
			#673 panFilterFailToRegen020104 <= filterFailToRegen020104
			#674 panErrorToOpenZD0204 <= errorToOpenZD0204
			#675 panErrorToCloseZD0204 <= errorToCloseZD0204
			#676 panErrorToOpenZD0210 <= errorToOpenZD0210
			#677 panErrorToCloseZD0210 <= errorToCloseZD0210
			#678 panFilterFailToRegen020105 <= filterFailToRegen020105
			#679 panErrorToOpenZD0205 <= errorToOpenZD0205
			#680 panErrorToCloseZD0205 <= errorToCloseZD0205
		END_MACRO
		#681 MACRO 8 bit output module 12()
			#682 panErrorToOpenZD0211 <= errorToOpenZD0211
			#683 panErrorToCloseZD0211 <= errorToCloseZD0211
			#684 panFilterFailToRegen020106 <= filterFailToRegen020106
			#685 panErrorToOpenZD0206 <= errorToOpenZD0206
			#686 panErrorToCloseZD0206 <= errorToCloseZD0206
			#687 panErrorToOpenZD0212 <= errorToOpenZD0212
			#688 panErrorToCloseZD0212 <= errorToCloseZD0212
			#689 panFilterFailToRegen020201 <= filterFailToRegen020201
		END_MACRO
		#690 MACRO 8 bit output module 13()
			#691 panErrorToOpenZD0213 <= errorToOpenZD0213
			#692 panErrorToCloseZD0213 <= errorToCloseZD0213
			#693 panErrorToOpenZD0219 <= errorToOpenZD0219
			#694 panErrorToCloseZD0219 <= errorToCloseZD0219
			#695 panFilterFailToRegen020202 <= filterFailToRegen020202
			#696 panErrorToOpenZD0214 <= errorToOpenZD0214
			#697 panErrorToCloseZD0214 <= errorToCloseZD0214
			#698 panErrorToOpenZD0220 <= errorToOpenZD0220
		END_MACRO
		#699 MACRO 8 bit output module 14()
			#700 panErrorToCloseZD0220 <= errorToCloseZD0220
			#701 panFilterFailToRegen020203 <= filterFailToRegen020203
			#702 panErrorToOpenZD0215 <= errorToOpenZD0215
			#703 panErrorToCloseZD0215 <= errorToCloseZD0215
			#704 panErrorToOpenZD0221 <= errorToOpenZD0221
			#705 panErrorToCloseZD0221 <= errorToCloseZD0221
			#706 panFilterFailToRegen020204 <= filterFailToRegen020204
			#707 panErrorToOpenZD0216 <= errorToOpenZD0216
		END_MACRO
		#708 MACRO 8 bit output module 15()
			#709 panErrorToCloseZD0216 <= errorToCloseZD0216
			#710 panErrorToOpenZD0222 <= errorToOpenZD0222
			#711 panErrorToCloseZD0222 <= errorToCloseZD0222
			#712 panFilterFailToRegen020205 <= filterFailToRegen020205
			#713 panErrorToOpenZD0217 <= errorToOpenZD0217
			#714 panErrorToCloseZD0217 <= errorToCloseZD0217
			#715 panErrorToOpenZD0223 <= errorToOpenZD0223
			#716 panErrorToCloseZD0223 <= errorToCloseZD0223
		END_MACRO
		#717 MACRO 8 bit output module 16()
			#718 panFilterFailToRegen020206 <= filterFailToRegen020206
			#719 panErrorToOpenZD0218 <= errorToOpenZD0218
			#720 panErrorToCloseZD0218 <= errorToCloseZD0218
			#721 panErrorToOpenZD0224 <= errorToOpenZD0224
			#722 panErrorToCloseZD0224 <= errorToCloseZD0224
			#723 panAlarmPLKnetwork <= alarmPLKnetwork
			#724 panAlarmND050201 <= alarmND050201
			#725 panAlarmND050202 <= alarmND050202
		END_MACRO
		#726 MACRO 8 bit output module 17()
			#727 panAlarmND060201 <= alarmND060201
			#728 panAlarmND060202 <= alarmND060202
			#729 panAlarmND060301 <= alarmND060301
			#730 panAlarmND060302 <= alarmND060302
			#731 panAlarmND070301 <= alarmND070301
			#732 panAlarmND070302 <= alarmND070302
			#733 panAlarmND080301 <= alarmND080301
			#734 panAlarmND080302 <= alarmND080302
		END_MACRO
		#735 MACRO 8 bit output module 18()
			#736 panAlarmND0804 <= alarmND0804
			#737 panAlarmOGM0104overload <= alarmOGM0104overload
			#738 panAlarmRCHV0203overload <= alarmRCHV0203overload
			#739 panAlarmN040402 <= alarmN040402
			#740 panAlarmN040401 <= alarmN040401
			#741 panAlarmM0604 <= alarmM0604
			#742 panAlarmM0702 <= alarmM0702
			#743 panAlarmM0802 <= alarmM0802
		END_MACRO
		#744 MACRO 8 bit output module 19()
			#745 panAlarmN020401 <= alarmN020401
			#746 panAlarmN020402 <= alarmN020402
			#747 panAlarmFS020101 <= alarmFS020101
			#748 panAlarmFS020102 <= alarmFS020102
			#749 panAlarmFS020103 <= alarmFS020103
			#750 panAlarmFS020104 <= alarmFS020104
			#751 panAlarmFS020105 <= alarmFS020105
			#752 panAlarmFS020106 <= alarmFS020106
		END_MACRO
		#753 MACRO 8 bit output module 20()
			#754 panAlarmFS020201 <= alarmFS020201
			#755 panAlarmFS020202 <= alarmFS020202
			#756 panAlarmFS020203 <= alarmFS020203
			#757 panAlarmFS020204 <= alarmFS020204
			#758 panAlarmFS020205 <= alarmFS020205
			#759 panAlarmFS020206 <= alarmFS020206
			#760 panAlarmZDE0201power <= alarmZDE0201power
			#761 panAlarmZDE0202power <= alarmZDE0202power
		END_MACRO
		#762 MACRO 8 bit output module 21()
			#763 panAlarmZDE0203power <= alarmZDE0203power
			#764 panAlarmZDE0204power <= alarmZDE0204power
			#765 panAlarmZDE0205power <= alarmZDE0205power
			#766 panAlarmZDE0206power <= alarmZDE0206power
			#767 panAlarmZDE0207power <= alarmZDE0207power
			#768 panAlarmZDE0208power <= alarmZDE0208power
			#769 panAlarmZDE0209power <= alarmZDE0209power
			#770 panAlarmZDE0210power <= alarmZDE0210power
		END_MACRO
		#771 MACRO 8 bit output module 22()
			#772 panAlarmZDE0211power <= alarmZDE0211power
			#773 panAlarmZDE0212power <= alarmZDE0212power
			#774 panAlarmZDE0213power <= alarmZDE0213power
			#775 panAlarmZDE0214power <= alarmZDE0214power
			#776 panAlarmZDE0215power <= alarmZDE0215power
			#777 panAlarmZDE0216power <= alarmZDE0216power
			#778 panAlarmZDE0217power <= alarmZDE0217power
			#779 panAlarmZDE0218power <= alarmZDE0218power
		END_MACRO
		#780 MACRO 8 bit output module 23()
			#781 panAlarmZDE0219power <= alarmZDE0219power
			#782 panAlarmZDE0220power <= alarmZDE0220power
			#783 panAlarmZDE0221power <= alarmZDE0221power
			#784 panAlarmZDE0222power <= alarmZDE0222power
			#785 panAlarmZDE0223power <= alarmZDE0223power
			#786 panAlarmZDE0224power <= alarmZDE0224power
			#787 panAlarmZDE0225power <= alarmZDE0225power
			#788 panAlarmKSHE0401power <= alarmKSHE0401power
		END_MACRO
		#789 MACRO 8 bit output module 24()
			#790 panAlarmKNS <= alarmKNS
			#791 panAlarmPowerSocketFS <= alarmPowerSocketFS
			#792 panAlarmKEMvalvesPower <= alarmKEMvalvesPower
			#793 panAlarmEmergencyPressed <= alarmEmergencyPressed
			#794 panAlarmRKF <= alarmRKF
			#795 panUFO0301noFlowAttention <= UFO0301noFlowAttention
			#796 panM0604attention <= M0604attention
			#797 panM0702attention <= M0702attention
		END_MACRO
		#798 MACRO 8 bit output module 25()
			#799 panM0802attention <= M0802attention
			#800 panStatusKNS <= DD6_DI.8
			#801 panND0502statRegimeP1M <= ND0502statRegimeP1M
			#802 panND0502statRegimeP2M <= ND0502statRegimeP2M
			#803 panND0502statRegimeByC <= ND0502statRegimeByC
			#804 panND0502statRegimeByWT <= ND0502statRegimeByWT
			#805 panND0602statRegimeP1M <= ND0602statRegimeP1M
			#806 panND0602statRegimeP2M <= ND0602statRegimeP2M
		END_MACRO
		#807 MACRO 8 bit output module 26()
			#808 panND0602statRegimeByC <= ND0602statRegimeByC
			#809 panND0602statRegimeByWT <= ND0602statRegimeByWT
			#810 panND0603statRegimeP1M <= ND0603statRegimeP1M
			#811 panND0603statRegimeP2M <= ND0603statRegimeP2M
			#812 panND0603statRegimeByC <= ND0603statRegimeByC
			#813 panND0603statRegimeByWT <= ND0603statRegimeByWT
			#814 panND0703statRegimeP1M <= ND0703statRegimeP1M
			#815 panND0703statRegimeP2M <= ND0703statRegimeP2M
		END_MACRO
		#816 MACRO 8 bit output module 27()
			#817 panND0703statRegimeByC <= ND0703statRegimeByC
			#818 panND0703statRegimeByWT <= ND0703statRegimeByWT
			#819 panND0803statRegimeP1M <= ND0803statRegimeP1M
			#820 panND0803statRegimeP2M <= ND0803statRegimeP2M
			#821 panND0803statRegimeByC <= ND0803statRegimeByC
			#822 panND0803statRegimeByWT <= ND0803statRegimeByWT
			#823 panN0105statRegimeP1M <= N0105statRegimeP1M
			#824 panN0105statRegimeP2M <= N0105statRegimeP2M
		END_MACRO
		#825 MACRO 8 bit output module 28()
			#826 panN0105statRegimeByC <= N0105statRegimeByC
			#827 panN0105statRegimeByWT <= N0105statRegimeByWT
			#828 panN0204statRegimeP1M <= N0204statRegimeP1M
			#829 panN0204statRegimeP2M <= N0204statRegimeP2M
			#830 panN0204statRegimeByC <= N0204statRegimeByC
			#831 panN0204statRegimeWT <= N0204statRegimeWT
			#832 panN0404statRegimeP1M <= N0404statRegimeP1M
			#833 panN0404statRegimeP2M <= N0404statRegimeP2M
		END_MACRO
		#834 MACRO 8 bit output module 29()
			#835 panN0404statRegimeByC <= N0404statRegimeByC
			#836 panN0404statRegimeWT <= N0404statRegimeWT
			#837 panUFO0301statRegimeP1M <= UFO0301statRegimeP1M
			#838 panUFO0301statRegimeP2M <= UFO0301statRegimeP2M
			#839 panUFO0301statRegimeByC <= UFO0301statRegimeByC
			#840 panUFO0301statRegimeWT <= UFO0301statRegimeWT
			#841 panZDE0225open <= DD9_DI.0
			#842 panZDE0201open <= DD7_DI.16
		END_MACRO
		#843 MACRO 8 bit output module 30()
			#844 panZDE0201close <= DD7_DI.17
			#845 panZDE0202open <= DD7_DI.18
			#846 panZDE0202close <= DD7_DI.19
			#847 panZDE0203open <= DD7_DI.20
			#848 panZDE0203close <= DD7_DI.21
			#849 panZDE0204open <= DD7_DI.22
			#850 panZDE0204close <= DD7_DI.23
			#851 panZDE0205open <= DD7_DI.24
		END_MACRO
		#852 MACRO 8 bit output module 31()
			#853 panZDE0205close <= DD7_DI.25
			#854 panZDE0206open <= DD7_DI.26
			#855 panZDE0206close <= DD7_DI.27
			#856 panZDE0207open <= DD7_DI.28
			#857 panZDE0207close <= DD7_DI.29
			#858 panZDE0208open <= DD7_DI.30
			#859 panZDE0208close <= DD7_DI.31
			#860 panZDE0209open <= DD8_DI.0
		END_MACRO
		#861 MACRO 8 bit output module 32()
			#862 panZDE0209close <= DD8_DI.1
			#863 panZDE0210open <= DD8_DI.2
			#864 panZDE0210close <= DD8_DI.3
			#865 panZDE0211open <= DD8_DI.4
			#866 panZDE0211close <= DD8_DI.5
			#867 panZDE0212open <= DD8_DI.6
			#868 panZDE0212close <= DD8_DI.7
			#869 panZDE0213open <= DD8_DI.8
		END_MACRO
		#870 MACRO 8 bit output module 33()
			#871 panZDE0213close <= DD8_DI.9
			#872 panZDE0214open <= DD8_DI.10
			#873 panZDE0214close <= DD8_DI.11
			#874 panZDE0215open <= DD8_DI.12
			#875 panZDE0215close <= DD8_DI.13
			#876 panZDE0216open <= DD8_DI.14
			#877 panZDE0216close <= DD8_DI.15
			#878 panZDE0217open <= DD8_DI.16
		END_MACRO
		#879 MACRO 8 bit output module 34()
			#880 panZDE0217close <= DD8_DI.17
			#881 panZDE0218open <= DD8_DI.18
			#882 panZDE0218close <= DD8_DI.19
			#883 panZDE0219open <= DD8_DI.20
			#884 panZDE0219close <= DD8_DI.21
			#885 panZDE0220open <= DD8_DI.22
			#886 panZDE0220close <= DD8_DI.23
			#887 panZDE0221open <= DD8_DI.24
		END_MACRO
		#888 MACRO 8 bit output module 35()
			#889 panZDE0221close <= DD8_DI.25
			#890 panZDE0222open <= DD8_DI.26
			#891 panZDE0222close <= DD8_DI.27
			#892 panZDE0223open <= DD8_DI.28
			#893 panZDE0223close <= DD8_DI.29
			#894 panZDE0224open <= DD8_DI.30
			#895 panZDE0224close <= DD8_DI.31
			#896 panZDE0225close <= DD9_DI.1
		END_MACRO
		#897 MACRO 8 bit output module 36x()
			#898 panKSHE0401close <= DD9_DI.3
			#899 panZDE0301open <= DD1_DI12
			#900 panZDE0301close <= DD1_DI13
			#901 panZDE0302open <= DD1_DI14
			#902 panZDE0302close <= DD1_DI15
			#903 panErrorToOpenZDE0301 <= errorToOpenZDE0301
			#904 panErrorToCloseZDE0301 <= errorToCloseZDE0301
			#905 panErrorToOpenZDE0302 <= errorToOpenZDE0302
		END_MACRO
		#906 panErrorToCloseZDE0302 <= errorToCloseZDE0302
		#907 panAlarmZDE0301power <= alarmZDE0301power
		#908 panAlarmZDE0302power <= alarmZDE0302power
		#909 panUFO030101danger <= statusUFO030101danger
		#910 panUFO030102danger <= statusUFO030102danger
		#911 panUFO030101distantMode <= statusUFO030101distantMode
		#912 panUFO030102distantMode <= statusUFO030102distantMode
	END_MACRO
	#913 MACRO PFW регистры на чтение из панели (управление ПЛК)()
		#914 MUL(panTimeToOpenCloseValve, 1000)
		#915 REAL_TO_TIME(#914)
		#916 TimeToOpenCloseValve <= #915
		#917 maxTemperature <= panMaxTemperature
		#918 minTemperature <= panMinTemperature
		#919 ND0502setMaxDosVal <= panND0502setMaxDosVal
		#920 ND0502setKoefProp <= panND0502setKoefProp
		#921 ND0602setMaxDosVal <= panND0602setMaxDosVal
		#922 ND0602setKoefProp <= panND0602setKoefProp
		#923 ND0603setMaxDosVal <= panND0603setMaxDosVal
		#924 ND0603setKoefProp <= panND0603setKoefProp
		#925 ND0703pHsetValue <= panND0703pHsetValue
		#926 ND0703YoutManual <= panND0703YoutManual
		#927 ND0703koeffI <= panND0703koeffI
		#928 ND0703koeffD <= panND0703koeffD
		#929 ND0703koeffP <= panND0703koeffP
		#930 ND0803setMaxDosVal <= panND0803setMaxDosVal
		#931 ND0803setKoefProp <= panND0803setKoefProp
		#932 ND0804doseValue <= panND0804doseValue
		#933 N0105flowSetValue <= panN0105flowSetValue
		#934 N0105YoutManual <= panN0105YoutManual
		#935 N0105koeffI <= panN0105koeffI
		#936 N0105koeffD <= panN0105koeffD
		#937 N0105koeffP <= panN0105koeffP
		#938 FQS0301impulsValue <= panFQS0301impulsValue
		#939 FQS0301correction <= panFQS0301correction
		#940 MUL(panFPKtimeToWork, 1000)
		#941 REAL_TO_TIME(#940)
		#942 FPKtimeToWork <= #941
		#943 MUL(panFPKnotStartedTime, 1000)
		#944 REAL_TO_TIME(#943)
		#945 FPKnotStartedTime <= #944
		#946 FPKmaxPressureValue <= panFPKmaxPressureValue
		#947 filterValueToRegen <= panFilterValueToRegen
	END_MACRO
	#948 MACRO PSB регистры на чтение из панели (управление ПЛК)()
		(* PSB регистры на чтение из панели (управление ПЛК) *)
		#949 MACRO 8 bit input module 1()
			#1279 alarmReset <= panAlarmResetButton
			#1280 ND0502resetCountP1 <= panND0502resetCountP1
			#1281 ND0502resetCountP2 <= panND0502resetCountP2
			#1282 ND0502resetWorkTimeP1 <= panND0502resetWorkTimeP1
			#1283 ND0502resetWorkTimeP2 <= panND0502resetWorkTimeP2
			#1284 ND0502regimeP1M <= panND0502regimeP1M
			#1285 ND0502regimeP2M <= panND0502regimeP2M
			#1286 ND0502regimeByC <= panND0502regimeByC
		END_MACRO
		#950 MACRO 8 bit input module 2()
			#1287 ND0502regimeByWT <= panND0502regimeByWT
			#1288 ND0602resetCountP1 <= panND0602resetCountP1
			#1289 ND0602resetCountP2 <= panND0602resetCountP2
			#1290 ND0602resetWorkTimeP1 <= panND0602resetWorkTimeP1
			#1291 ND0602resetWorkTimeP2 <= panND0602resetWorkTimeP2
			#1292 ND0602regimeP1M <= panND0602regimeP1M
			#1293 ND0602regimeP2M <= panND0602regimeP2M
			#1294 ND0602regimeByC <= panND0602regimeByC
		END_MACRO
		#951 MACRO 8 bit input module 3()
			#1295 ND0602regimeByWT <= panND0602regimeByWT
			#1296 ND0603resetCountP1 <= panND0603resetCountP1
			#1297 ND0603resetCountP2 <= panND0603resetCountP2
			#1298 ND0603resetWorkTimeP1 <= panND0603resetWorkTimeP1
			#1299 ND0603resetWorkTimeP2 <= panND0603resetWorkTimeP2
			#1300 ND0603regimeP1M <= panND0603regimeP1M
			#1301 ND0603regimeP2M <= panND0603regimeP2M
			#1302 ND0603regimeByC <= panND0603regimeByC
		END_MACRO
		#952 MACRO 8 bit input module 4()
			#1303 ND0603regimeByWT <= panND0603regimeByWT
			#1304 ND0703resetCountP1 <= panND0703resetCountP1
			#1305 ND0703resetCountP2 <= panND0703resetCountP2
			#1306 ND0703resetWorkTimeP1 <= panND0703resetWorkTimeP1
			#1307 ND0703resetWorkTimeP2 <= panND0703resetWorkTimeP2
			#1308 ND0703regimeP1M <= panND0703regimeP1M
			#1309 ND0703regimeP2M <= panND0703regimeP2M
			#1310 ND0703regimeByC <= panND0703regimeByC
		END_MACRO
		#953 MACRO 8 bit input module 5()
			#1311 ND0703regimeByWT <= panND0703regimeByWT
			#1312 ND0703YmanAuto <= panND0703YmanAuto
			#1313 ND0803resetCountP1 <= panND0803resetCountP1
			#1314 ND0803resetCountP2 <= panND0803resetCountP2
			#1315 ND0803resetWorkTimeP1 <= panND0803resetWorkTimeP1
			#1316 ND0803resetWorkTimeP2 <= panND0803resetWorkTimeP2
			#1317 ND0803regimeP1M <= panND0803regimeP1M
			#1318 ND0803regimeP2M <= panND0803regimeP2M
		END_MACRO
		#954 MACRO 8 bit input module 6()
			#1319 ND0803regimeByC <= panND0803regimeByC
			#1320 ND0803regimeByWT <= panND0803regimeByWT
			#1321 N0105resetCountP1 <= panN0105resetCountP1
			#1322 N0105resetCountP2 <= panN0105resetCountP2
			#1323 N0105resetWorkTimeP1 <= panN0105resetWorkTimeP1
			#1324 N0105resetWorkTimeP2 <= panN0105resetWorkTimeP2
			#1325 N0105regimeByC <= panN0105regimeByC
			#1326 N0105regimeByWT <= panN0105regimeByWT
		END_MACRO
		#955 MACRO 8 bit input module 7()
			#1327 N0105YmanAuto <= panN0105YmanAuto
			#1328 N0204resetCountP1 <= panN0204resetCountP1
			#1329 N0204resetCountP2 <= panN0204resetCountP2
			#1330 N0204resetWorkTimeP1 <= panN0204resetWorkTimeP1
			#1331 N0204resetWorkTimeP2 <= panN0204resetWorkTimeP2
			#1332 N0204regimeP1M <= panN0204regimeP1M
			#1333 N0204regimeP2M <= panN0204regimeP2M
			#1334 N0204regimeByC <= panN0204regimeByC
		END_MACRO
		#956 MACRO 8 bit input module 8()
			#1335 N0204regimeWT <= panN0204regimeWT
			#1336 UFO0301resetCountP1 <= panUFO0301resetCountP1
			#1337 UFO0301resetCountP2 <= panUFO0301resetCountP2
			#1338 UFO0301resetWorkTimeP1 <= panUFO0301resetWorkTimeP1
			#1339 UFO0301resetWorkTimeP2 <= panUFO0301resetWorkTimeP2
			#1340 UFO0301regimeP1M <= panUFO0301regimeP1M
			#1341 UFO0301regimeP2M <= panUFO0301regimeP2M
			#1342 UFO0301regimeByC <= panUFO0301regimeByC
		END_MACRO
		#957 MACRO 8 bit input module 9()
			#1343 UFO0301regimeWT <= panUFO0301regimeWT
			#1344 N0404resetCountP1 <= panN0404resetCountP1
			#1345 N0404resetCountP2 <= panN0404resetCountP2
			#1346 N0404resetWorkTimeP1 <= panN0404resetWorkTimeP1
			#1347 N0404resetWorkTimeP2 <= panN0404resetWorkTimeP2
			#1348 N0404regimeP1M <= panN0404regimeP1M
			#1349 N0404regimeP2M <= panN0404regimeP2M
			#1350 N0404regimeByC <= panN0404regimeByC
		END_MACRO
		#958 MACRO 8 bit input module 10-11()
			(* одули 10 и 11 заполнены переменными для тестирования задвижек. / Здесь они не показаны, т.к. спешка. / Они вставлены напрямую в макросы управления промывкой фильтров. / testValvesFS020101 - testValvesFS020206 (PSB612-623) *)
			#1351 N0404regimeWT <= panN0404regimeWT
			#1352 FQS0301reset <= panFQS0301reset
			#1353 FQS0301addCorrection <= panFQS0301addCorrection
			#1354 FQS0301deleteCorrection <= panFQS0301deleteCorrection
		END_MACRO
		#959 testKSHE0401 <= panTestKSHE0401
		#960 testZDE0225 <= panTestZDE0225
		#961 testZDE03 <= panTestZDE03
		#962 manualZDE0301 <= panManualZDE0301
		#963 manualZDE0302 <= panManualZDE0302
	END_MACRO
END_MACRO
#964 NOT(DD6_DI.13)
#965 alarmRCHV0203overload <= #964
#966 NOT(DD9_DI.5)
#967 alarmZDE0202power <= #966
#968 NOT(DD9_DI.26)
#969 alarmZDE0223power <= #968
#970 MACRO переменные на диспетчеризацию()
	#971 remFT0101value <= DD1_AI1_FT0101value
	#972 remFQS0301totalAmount <= FQS0301totalAmount
	#973 remTemperatureValue <= temperatureValue
	#974 remStatusN010501started <= N0105statStartedP1
	#975 remStatusN010502started <= N0105statStartedP2
	#976 remStatusUFO030101started <= statusUFO030101started
	#977 remStatusUFO030102started <= statusUFO030102started
	#978 remAlarm <= Alarm
	#979 remN010501alarm <= N010501alarm
	#980 remN010502alarm <= N010502alarm
	#981 remFPKalarm <= DD7_DI.14
	#982 remUFO030101alarm <= statusUFO030101alarm
	#983 remUFO030102alarm <= statusUFO030102alarm
	#984 remAlarmEmergencyPressed <= alarmEmergencyPressed
	#985 remAlarmOOGM0104overload <= DD6_DI.11
	#986 remAlarmRCHV0203overload <= DD6_DI.13
END_MACRO
#987 NOT(DD5_DI.14)
#988 alarmN040402 <= #987
#989 NOT(DD9_DI.6)
#990 alarmZDE0203power <= #989
#991 NOT(DD9_DI.27)
#992 alarmZDE0224power <= #991
#993 NOT(DD5_DI.15)
#994 alarmN040401 <= #993
#995 NOT(DD9_DI.7)
#996 alarmZDE0204power <= #995
#997 NOT(DD9_DI.28)
#998 alarmZDE0225power <= #997
#999 NOT(DD5_DI.20)
#1000 alarmM0604 <= #999
#1001 NOT(DD9_DI.8)
#1002 alarmZDE0205power <= #1001
#1003 NOT(DD9_DI.29)
#1004 alarmKSHE0401power <= #1003
#1005 NOT(DD5_DI.22)
#1006 alarmM0702 <= #1005
#1007 NOT(DD9_DI.9)
#1008 alarmZDE0206power <= #1007
#1009 NOT(DD6_DI.9)
#1010 alarmKNS <= #1009
#1011 NOT(DD5_DI.24)
#1012 alarmM0802 <= #1011
#1013 NOT(DD9_DI.10)
#1014 alarmZDE0207power <= #1013
#1015 NOT(DD6_DI.17)
#1016 alarmPowerSocketFS <= #1015
#1017 NOT(DD5_DI.7)
#1018 alarmN020401 <= #1017
#1019 NOT(DD9_DI.11)
#1020 alarmZDE0208power <= #1019
#1021 NOT(DD6_DI.18)
#1022 alarmKEMvalvesPower <= #1021
#1023 NOT(DD5_DI.8)
#1024 alarmN020402 <= #1023
#1025 NOT(DD9_DI.12)
#1026 alarmZDE0209power <= #1025
#1027 NOT(DD1_DI4)
#1028 alarmEmergencyPressed <= #1027
#1029 GT(DD1_AI2_FT0102value, 0)
#1030 filterPulserGen:PulsePerSec(start: #1029)
#1031 DIV(DD1_AI2_FT0102value, 3600)
#1032 ADD(EN: #1030.out, #1031, filterTotalAmountFT0102)
#1033 filterTotalAmountFT0102 <= #1032
#1034 NOT(DD6_DI.21)
#1035 alarmFS020101 <= #1034
#1036 NOT(DD9_DI.13)
#1037 alarmZDE0210power <= #1036
#1038 NOT(DD1_DI5)
#1039 alarmRKF <= #1038
#1040 NOT(DD9_DI.30)
#1041 alarmZDE0301power <= #1040
#1042 NOT(DD9_DI.31)
#1043 alarmZDE0302power <= #1042
#1044 MOVE(EN: filterTotalAmountReset, 0)
#1045 filterTotalAmountFT0102 <= #1044
#1046 SUB(filterValueToRegen, filterTotalAmountFT0102)
#1047 volumeToRegen <= #1046
#1048 GE(filterTotalAmountFT0102, filterValueToRegen)
#1049 MACRO управление промывкой фильтра ФС02.01.01(pin 1 "сигнал на промывку": #1048, pin 2 "авария фильтра": DD6_DI.21, pin 3 "подтверждение промывки": DD6_DI.20, pin 4 "сброс аварий": alarmReset, pin 5 "начать очередь снова": filterStartNewQueue, pin 6 "ЗДЭ02.01 открыта": DD7_DI.16, pin 7 "ЗДЭ02.01 закрыта": DD7_DI.17, pin 8 "ЗДЭ02.07 открыта": DD7_DI.28, pin 9 "ЗДЭ02.07 закрыта": DD7_DI.29, pin 10 "время движения ЗДЭ": timeToOpenCloseValve, pin 11 "авария питания ЗДЭ02.01": DD9_DI.4, pin 12 "авария питания ЗДЭ02.07": DD9_DI.10)
	(* если открыт = фильтрация *)
	(* если открыт = промывка *)
	(* <- выход использовать в / последнем фильтре для / начала очереди заново *)
	out 1 "следующий в очереди" <= #1052.output
	out 2 "промыть ФС02.01.01" <= #1051
	#1050 ZD0201:SimpleValve(inputOpen: NOT #1051, inputClose: #1051, statusOpen: pin 6, statusClose: pin 7, reset: pin 4, timeToOpenClose: pin 10)
	out 6 "открыть ЗДЭ02.01" <= #1050.outputOpen
	out 7 "закрыть ЗДЭ02.01" <= #1050.outputClose
	out 8 "авария открытия ЗДЭ02.01" <= #1050.errorToOpen
	#1051 OR(panTestValvesFS020101, #1052.regenFilterOUT)
	out 9 "авария закрытия ЗДЭ02.01" <= #1050.errorToClose
	#1052 FS020101manager:FilterQueueManager(input: pin 1, filterAlarm: #1053, regenFilterStatus: pin 3, alarmReset: pin 4, startNextLoop: pin 5)
	#1053 OR(alarmZD020107, pin 2, pin 11, pin 12)
	out 3 "ФС02.01.01 промыт" <= #1052.regenerated
	out 4 "не удалось промыть" <= #1052.failToRegen
	#1054 OR(#1050.errorToOpen, #1050.errorToClose, #1056.errorToOpen, #1056.errorToClose)
	#1055 alarmZD020107 <= #1054
	out 5 "сброс счетчика" <= #1052.counterReset
	#1056 ZD0207:SimpleValve(inputOpen: #1051, inputClose: NOT #1051, statusOpen: pin 8, statusClose: pin 9, reset: pin 4, timeToOpenClose: pin 10)
	out 10 "открыть ЗДЭ02.07" <= #1056.outputOpen
	out 11 "закрыть ЗДЭ02.07" <= #1056.outputClose
	out 12 "авария открытия ЗДЭ02.07" <= #1056.errorToOpen
	out 13 "авария закрытия ЗДЭ02.07" <= #1056.errorToClose
END_MACRO
#1057 DD2_DO.4 <= #1049.out 2
#1058 regeneratedFS020101 <= #1049.out 3
#1059 filterFailToRegen020101 <= #1049.out 4
#1060 filterTotalAmountReset <= #1049.out 5
#1061 DD2_DO.16 <= #1049.out 6
#1062 DD2_DO.17 <= #1049.out 7
#1063 errorToOpenZD0201 <= #1049.out 8
#1064 errorToCloseZD0201 <= #1049.out 9
#1065 DD2_DO.28 <= #1049.out 10
#1066 DD2_DO.29 <= #1049.out 11
#1067 errorToOpenZD0207 <= #1049.out 12
#1068 errorToCloseZD0207 <= #1049.out 13
#1069 MACRO управление промывкой фильтра ФС02.01.02(pin 1 "сигнал на промывку": #1049.out 1, pin 2 "авария фильтра": DD6_DI.23, pin 3 "подтверждение промывки": DD6_DI.22, pin 4 "сброс аварий": alarmReset, pin 5 "начать очередь снова": filterStartNewQueue, pin 6 "ЗДЭ02.02 открыта": DD7_DI.18, pin 7 "ЗДЭ02.02 закрыта": DD7_DI.19, pin 8 "ЗДЭ02.08 открыта": DD7_DI.30, pin 9 "ЗДЭ02.08 закрыта": DD7_DI.31, pin 10 "время движения ЗДЭ": timeToOpenCloseValve, pin 11 "авария питания ЗДЭ02.02": DD9_DI.5, pin 12 "авария питания ЗДЭ02.08": DD9_DI.11)
	(* если открыт = фильтрация *)
	(* если открыт = промывка *)
	(* <- выход использовать в / последнем фильтре для / начала очереди заново *)
	out 1 "следующий в очереди" <= #1072.output
	out 2 "промыть ФС02.01.02" <= #1071
	#1070 ZD0202:SimpleValve(inputOpen: NOT #1071, inputClose: #1071, statusOpen: pin 6, statusClose: pin 7, reset: pin 4, timeToOpenClose: pin 10)
	out 5 "открыть ЗДЭ02.02" <= #1070.outputOpen
	out 6 "закрыть ЗДЭ02.02" <= #1070.outputClose
	out 7 "авария открытия ЗДЭ02.02" <= #1070.errorToOpen
	#1071 OR(panTestValvesFS020102, #1072.regenFilterOUT)
	out 8 "авария закрытия ЗДЭ02.02" <= #1070.errorToClose
	#1072 FS020102manager:FilterQueueManager(input: pin 1, filterAlarm: #1073, regenFilterStatus: pin 3, alarmReset: pin 4, startNextLoop: pin 5)
	#1073 OR(alarmZD020208, pin 2, pin 11, pin 12)
	#1074 OR(#1070.errorToOpen, #1070.errorToClose, #1076.errorToOpen, #1076.errorToClose)
	#1075 alarmZD020208 <= #1074
	out 3 "ФС02.01.02 промыт" <= #1072.regenerated
	out 4 "не удалось промыть" <= #1072.failToRegen
	#1076 ZD0208:SimpleValve(inputOpen: #1071, inputClose: NOT #1071, statusOpen: pin 8, statusClose: pin 9, reset: pin 4, timeToOpenClose: pin 10)
	out 9 "открыть ЗДЭ02.08" <= #1076.outputOpen
	out 10 "закрыть ЗДЭ02.08" <= #1076.outputClose
	out 11 "авария открытия ЗДЭ02.08" <= #1076.errorToOpen
	out 12 "авария закрытия ЗДЭ02.08" <= #1076.errorToClose
END_MACRO
#1077 DD2_DO.5 <= #1069.out 2
#1078 regeneratedFS020102 <= #1069.out 3
#1079 filterFailToRegen020102 <= #1069.out 4
#1080 DD2_DO.18 <= #1069.out 5
#1081 DD2_DO.19 <= #1069.out 6
#1082 errorToOpenZD0202 <= #1069.out 7
#1083 errorToCloseZD0202 <= #1069.out 8
#1084 DD2_DO.30 <= #1069.out 9
#1085 DD2_DO.31 <= #1069.out 10
#1086 errorToOpenZD0208 <= #1069.out 11
#1087 errorToCloseZD0208 <= #1069.out 12
#1088 MACRO управление промывкой фильтра ФС02.01.03(pin 1 "сигнал на промывку": #1069.out 1, pin 2 "авария фильтра": DD6_DI.25, pin 3 "подтверждение промывки": DD6_DI.24, pin 4 "сброс аварий": alarmReset, pin 5 "начать очередь снова": filterStartNewQueue, pin 6 "ЗДЭ02.03 открыта": DD7_DI.20, pin 7 "ЗДЭ02.03 закрыта": DD7_DI.21, pin 8 "ЗДЭ02.09 открыта": DD8_DI.0, pin 9 "ЗДЭ02.09 закрыта": DD8_DI.1, pin 10 "время движения ЗДЭ": timeToOpenCloseValve, pin 11 "авария питания ЗДЭ02.03": DD9_DI.6, pin 12 "авария питания ЗДЭ02.09": DD9_DI.12)
	(* если открыт = фильтрация *)
	(* если открыт = промывка *)
	(* <- выход использовать в / последнем фильтре для / начала очереди заново *)
	out 1 "следующий в очереди" <= #1091.output
	out 2 "промыть ФС02.01.03" <= #1090
	#1089 ZD0203:SimpleValve(inputOpen: NOT #1090, inputClose: #1090, statusOpen: pin 6, statusClose: pin 7, reset: pin 4, timeToOpenClose: pin 10)
	out 5 "открыть ЗДЭ02.03" <= #1089.outputOpen
	out 6 "закрыть ЗДЭ02.03" <= #1089.outputClose
	out 7 "авария открытия ЗДЭ02.03" <= #1089.errorToOpen
	#1090 OR(panTestValvesFS020103, #1091.regenFilterOUT)
	out 8 "авария закрытия ЗДЭ02.03" <= #1089.errorToClose
	#1091 FS020103manager:FilterQueueManager(input: pin 1, filterAlarm: #1092, regenFilterStatus: pin 3, alarmReset: pin 4, startNextLoop: pin 5)
	#1092 OR(alarmZD020309, pin 2, pin 11, pin 12)
	#1093 OR(#1089.errorToOpen, #1089.errorToClose, #1095.errorToOpen, #1095.errorToClose)
	#1094 alarmZD020309 <= #1093
	out 3 "ФС02.01.03 промыт" <= #1091.regenerated
	out 4 "не удалось промыть" <= #1091.failToRegen
	#1095 ZD0209:SimpleValve(inputOpen: #1090, inputClose: NOT #1090, statusOpen: pin 8, statusClose: pin 9, reset: pin 4, timeToOpenClose: pin 10)
	out 9 "открыть ЗДЭ02.09" <= #1095.outputOpen
	out 10 "закрыть ЗДЭ02.09" <= #1095.outputClose
	out 11 "авария открытия ЗДЭ02.09" <= #1095.errorToOpen
	out 12 "авария закрытия ЗДЭ02.09" <= #1095.errorToClose
END_MACRO
#1096 DD2_DO.6 <= #1088.out 2
#1097 regeneratedFS020103 <= #1088.out 3
#1098 filterFailToRegen020103 <= #1088.out 4
#1099 DD2_DO.20 <= #1088.out 5
#1100 DD2_DO.21 <= #1088.out 6
#1101 errorToOpenZD0203 <= #1088.out 7
#1102 errorToCloseZD0203 <= #1088.out 8
#1103 DD3_DO.0 <= #1088.out 9
#1104 DD3_DO.1 <= #1088.out 10
#1105 errorToOpenZD0209 <= #1088.out 11
#1106 errorToCloseZD0209 <= #1088.out 12
#1107 MACRO управление промывкой фильтра ФС02.01.04(pin 1 "сигнал на промывку": #1088.out 1, pin 2 "авария фильтра": DD6_DI.27, pin 3 "подтверждение промывки": DD6_DI.26, pin 4 "сброс аварий": alarmReset, pin 5 "начать очередь снова": filterStartNewQueue, pin 6 "ЗДЭ02.04 открыта": DD7_DI.22, pin 7 "ЗДЭ02.04 закрыта": DD7_DI.23, pin 8 "ЗДЭ02.10 открыта": DD8_DI.2, pin 9 "ЗДЭ02.10 закрыта": DD8_DI.3, pin 10 "время движения ЗДЭ": timeToOpenCloseValve, pin 11 "авария питания ЗДЭ02.04": DD9_DI.7, pin 12 "авария питания ЗДЭ02.10": DD9_DI.13)
	(* если открыт = фильтрация *)
	(* если открыт = промывка *)
	(* <- выход использовать в / последнем фильтре для / начала очереди заново *)
	out 1 "следующий в очереди" <= #1110.output
	out 2 "промыть ФС02.01.04" <= #1109
	#1108 ZD0204:SimpleValve(inputOpen: NOT #1109, inputClose: #1109, statusOpen: pin 6, statusClose: pin 7, reset: pin 4, timeToOpenClose: pin 10)
	out 5 "открыть ЗДЭ02.04" <= #1108.outputOpen
	out 6 "закрыть ЗДЭ02.04" <= #1108.outputClose
	out 7 "авария открытия ЗДЭ02.04" <= #1108.errorToOpen
	#1109 OR(panTestValvesFS020104, #1110.regenFilterOUT)
	out 8 "авария закрытия ЗДЭ02.04" <= #1108.errorToClose
	#1110 FS020104manager:FilterQueueManager(input: pin 1, filterAlarm: #1111, regenFilterStatus: pin 3, alarmReset: pin 4, startNextLoop: pin 5)
	#1111 OR(alarmZD020410, pin 2, pin 11, pin 12)
	#1112 OR(#1108.errorToOpen, #1108.errorToClose, #1114.errorToOpen, #1114.errorToClose)
	#1113 alarmZD020410 <= #1112
	out 3 "ФС02.01.04 промыт" <= #1110.regenerated
	out 4 "не удалось промыть" <= #1110.failToRegen
	#1114 ZD0210:SimpleValve(inputOpen: #1109, inputClose: NOT #1109, statusOpen: pin 8, statusClose: pin 9, reset: pin 4, timeToOpenClose: pin 10)
	out 9 "открыть ЗДЭ02.10" <= #1114.outputOpen
	out 10 "закрыть ЗДЭ02.10" <= #1114.outputClose
	out 11 "авария открытия ЗДЭ02.10" <= #1114.errorToOpen
	out 12 "авария закрытия ЗДЭ02.10" <= #1114.errorToClose
END_MACRO
#1115 DD2_DO.7 <= #1107.out 2
#1116 regeneratedFS020104 <= #1107.out 3
#1117 filterFailToRegen020104 <= #1107.out 4
#1118 DD2_DO.22 <= #1107.out 5
#1119 DD2_DO.23 <= #1107.out 6
#1120 errorToOpenZD0204 <= #1107.out 7
#1121 errorToCloseZD0204 <= #1107.out 8
#1122 DD3_DO.2 <= #1107.out 9
#1123 DD3_DO.3 <= #1107.out 10
#1124 errorToOpenZD0210 <= #1107.out 11
#1125 errorToCloseZD0210 <= #1107.out 12
#1126 MACRO управление промывкой фильтра ФС02.01.05(pin 1 "сигнал на промывку": #1107.out 1, pin 2 "авария фильтра": DD6_DI.29, pin 3 "подтверждение промывки": DD6_DI.28, pin 4 "сброс аварий": alarmReset, pin 5 "начать очередь снова": filterStartNewQueue, pin 6 "ЗДЭ02.05 открыта": DD7_DI.24, pin 7 "ЗДЭ02.05 закрыта": DD7_DI.25, pin 8 "ЗДЭ02.11 открыта": DD8_DI.4, pin 9 "ЗДЭ02.11 закрыта": DD8_DI.5, pin 10 "время движения ЗДЭ": timeToOpenCloseValve, pin 11 "авария питания ЗДЭ02.05": DD9_DI.8, pin 12 "авария питания ЗДЭ02.11": DD9_DI.14)
	(* если открыт = фильтрация *)
	(* если открыт = промывка *)
	(* <- выход использовать в / последнем фильтре для / начала очереди заново *)
	out 1 "следующий в очереди" <= #1129.output
	out 2 "промыть ФС02.01.05" <= #1128
	#1127 ZD0205:SimpleValve(inputOpen: NOT #1128, inputClose: #1128, statusOpen: pin 6, statusClose: pin 7, reset: pin 4, timeToOpenClose: pin 10)
	out 5 "открыть ЗДЭ02.05" <= #1127.outputOpen
	out 6 "закрыть ЗДЭ02.05" <= #1127.outputClose
	out 7 "авария открытия ЗДЭ02.05" <= #1127.errorToOpen
	#1128 OR(panTestValvesFS020105, #1129.regenFilterOUT)
	out 8 "авария закрытия ЗДЭ02.05" <= #1127.errorToClose
	#1129 FS020105manager:FilterQueueManager(input: pin 1, filterAlarm: #1130, regenFilterStatus: pin 3, alarmReset: pin 4, startNextLoop: pin 5)
	#1130 OR(alarmZD020511, pin 2, pin 11, pin 12)
	#1131 OR(#1127.errorToOpen, #1127.errorToClose, #1133.errorToOpen, #1133.errorToClose)
	#1132 alarmZD020511 <= #1131
	out 3 "ФС02.01.05 промыт" <= #1129.regenerated
	out 4 "не удалось промыть" <= #1129.failToRegen
	#1133 ZD0211:SimpleValve(inputOpen: #1128, inputClose: NOT #1128, statusOpen: pin 8, statusClose: pin 9, reset: pin 4, timeToOpenClose: pin 10)
	out 9 "открыть ЗДЭ02.11" <= #1133.outputOpen
	out 10 "закрыть ЗДЭ02.11" <= #1133.outputClose
	out 11 "авария открытия ЗДЭ02.11" <= #1133.errorToOpen
	out 12 "авария закрытия ЗДЭ02.11" <= #1133.errorToClose
END_MACRO
#1134 DD2_DO.8 <= #1126.out 2
#1135 regeneratedFS020105 <= #1126.out 3
#1136 filterFailToRegen020105 <= #1126.out 4
#1137 DD2_DO.24 <= #1126.out 5
#1138 DD2_DO.25 <= #1126.out 6
#1139 errorToOpenZD0205 <= #1126.out 7
#1140 errorToCloseZD0205 <= #1126.out 8
#1141 DD3_DO.4 <= #1126.out 9
#1142 DD3_DO.5 <= #1126.out 10
#1143 errorToOpenZD0211 <= #1126.out 11
#1144 errorToCloseZD0211 <= #1126.out 12
#1145 MACRO управление промывкой фильтра ФС02.01.06(pin 1 "сигнал на промывку": #1126.out 1, pin 2 "авария фильтра": DD6_DI.31, pin 3 "подтверждение промывки": DD6_DI.30, pin 4 "сброс аварий": alarmReset, pin 5 "начать очередь снова": filterStartNewQueue, pin 6 "ЗДЭ02.06 открыта": DD7_DI.26, pin 7 "ЗДЭ02.06 закрыта": DD7_DI.27, pin 8 "ЗДЭ02.12 открыта": DD8_DI.6, pin 9 "ЗДЭ02.12 закрыта": DD8_DI.7, pin 10 "время движения ЗДЭ": timeToOpenCloseValve, pin 11 "авария питания ЗДЭ02.06": DD9_DI.9, pin 12 "авария питания ЗДЭ02.12": DD9_DI.15)
	(* если открыт = фильтрация *)
	(* если открыт = промывка *)
	(* <- выход использовать в / последнем фильтре для / начала очереди заново *)
	out 1 "следующий в очереди" <= #1148.output
	out 2 "промыть ФС02.01.06" <= #1147
	#1146 ZD0206:SimpleValve(inputOpen: NOT #1147, inputClose: #1147, statusOpen: pin 6, statusClose: pin 7, reset: pin 4, timeToOpenClose: pin 10)
	out 5 "открыть ЗДЭ02.06" <= #1146.outputOpen
	out 6 "закрыть ЗДЭ02.06" <= #1146.outputClose
	out 7 "авария открытия ЗДЭ02.06" <= #1146.errorToOpen
	#1147 OR(panTestValvesFS020106, #1148.regenFilterOUT)
	out 8 "авария закрытия ЗДЭ02.06" <= #1146.errorToClose
	#1148 FS020106manager:FilterQueueManager(input: pin 1, filterAlarm: #1149, regenFilterStatus: pin 3, alarmReset: pin 4, startNextLoop: pin 5)
	#1149 OR(alarmZD020612, pin 2, pin 11, pin 12)
	#1150 OR(#1146.errorToOpen, #1146.errorToClose, #1152.errorToOpen, #1152.errorToClose)
	#1151 alarmZD020612 <= #1150
	out 3 "ФС02.01.06 промыт" <= #1148.regenerated
	out 4 "не удалось промыть" <= #1148.failToRegen
	#1152 ZD0212:SimpleValve(inputOpen: #1147, inputClose: NOT #1147, statusOpen: pin 8, statusClose: pin 9, reset: pin 4, timeToOpenClose: pin 10)
	out 9 "открыть ЗДЭ02.12" <= #1152.outputOpen
	out 10 "закрыть ЗДЭ02.12" <= #1152.outputClose
	out 11 "авария открытия ЗДЭ02.12" <= #1152.errorToOpen
	out 12 "авария закрытия ЗДЭ02.12" <= #1152.errorToClose
END_MACRO
#1153 DD2_DO.9 <= #1145.out 2
#1154 regeneratedFS020106 <= #1145.out 3
#1155 filterFailToRegen020106 <= #1145.out 4
#1156 DD2_DO.26 <= #1145.out 5
#1157 DD2_DO.27 <= #1145.out 6
#1158 errorToOpenZD0206 <= #1145.out 7
#1159 errorToCloseZD0206 <= #1145.out 8
#1160 DD3_DO.6 <= #1145.out 9
#1161 DD3_DO.7 <= #1145.out 10
#1162 errorToOpenZD0212 <= #1145.out 11
#1163 errorToCloseZD0212 <= #1145.out 12
